# B&R Automation Studio project Nitto
Automation Studio 4.0.14.208

## Configuration Config1

CPU , AutomationRuntime G4.06, Build 4.1.2, Safety 1.5

### Task classes (Cpu.sw)
```
Cyclic#1:
  ncsdcctrl <- MainMachineCtrl.ncsdcctrl.prg
  WebControl <- (binary)
Cyclic#2:
  dummy <- MainMachineCtrl.dummy.prg
  MAIN <- MainMachineCtrl.MAIN.prg
Cyclic#4:
  VisuTasks <- Visualization.VisuCycl.VisuTasks.prg
  VisuPages <- Visualization.VisuCycl.VisuPages.prg
  VisuRange <- Visualization.VisuCycl.VisuRange.prg
  GeneralAla <- Alarme.GeneralAlarms.prg
  al_hdl <- pkgRecipe.al_hdl.prg
Cyclic#8:
  picctrl <- pkgRecipe.picctrl.prg
  tool_hdl <- pkgRecipe.tool_hdl.prg
  csv_hdl <- pkgRecipe.csv_hdl.prg
  save2USB <- pkgRecipe.save2USB.prg
DataObjects: Acp10sys
NcDataObjects: acp10etxde <- acp10etxde.dob, gunwfeedi <- AxisObj.gunwfeedi.dob, gunwfeeda <- AxisObj.gunwfeeda.dob, gmasteri <- AxisObj.gmasteri.dob, gpbs1i <- AxisObj.gpbs1i.dob, gpbs2i <- AxisObj.gpbs2i.dob, gcut1i <- AxisObj.gcut1i.dob, gcut2i <- AxisObj.gcut2i.dob, gunwopi <- AxisObj.gunwopi.dob, gunwdrvi <- AxisObj.gunwdrvi.dob, ggrid1i <- AxisObj.ggrid1i.dob, ggrid2i <- AxisObj.ggrid2i.dob, gbufferi <- AxisObj.gbufferi.dob, glongcuti <- AxisObj.glongcuti.dob, gcatchbi <- AxisObj.gcatchbi.dob, ggridfeedi <- AxisObj.ggridfeedi.dob, gconvbi <- AxisObj.gconvbi.dob, gbuffera <- AxisObj.gbuffera.dob, ggrida <- AxisObj.ggrida.dob, gunwa <- AxisObj.gunwa.dob, gpbs1a <- AxisObj.gpbs1a.dob, gpbs2a <- AxisObj.gpbs2a.dob, gcatchba <- AxisObj.gcatchba.dob, gsafetya <- AxisObj.gsafetya.dob, gconvbelta <- AxisObj.gconvbelta.dob, acp10etxd1 <- acp10etxde.dob, gPackBelta <- AxisObj.gPackBelta.dob, gPackBelti <- AxisObj.gPackBelti.dob, gCut1, gCut2, ggridfeede
VcDataObjects: Visu <- Visualization.VisuCycl.Visu.dob, Visu1 <- Visualization.VisuCycl.Visu1.dob, Visu2 <- Visualization.VisuCycl.Visu2.dob
Binaries: vcpkat, vcnet, vcpdvnc, vccpopup, vcclbox, vcctext, vccovl, vccalarm, Visu03, vccnum, vcchspot, arialbd, vccline, vccbtn, vccstr, vccddbox, vccbmp, vccshape, vccdt, vcfile, arial, vctcal, vcshared, vcrt, vcmgr, vcbclass, Visu02, vcgclass, vcdsint, vcptelo, Visu01, vcpdsw, vcpfapc, vcresman, vcpdi855, vcpdi815, vcfntttf, vcalarm, vcdsloc, vcpfmtcx, visvc, Visu103, vcpdihd, Visu102, vcpfpp50, Visu101, vcvisapi, Visu202, vcchtml, Visu201, vccurl, vcxml, Visu203, acp10cfg, acp10map, asfw, iomap, arconfig, sysconf, ashwd
Libraries: Acp10man, Acp10par, NcGlobal, UtilTyp, AsARCfg, AsBrMath, AsBrStr, AsMem, asstring, AsUSB, brsystem, FileIO, LoopConR, powerlnk, standard, sys_lib, Visapi, CSV_File, HlpStr, SwitchConf, TorqueCtrl, UserVC, Acp10_MC, Acp10sdc, SafeMC, MC_RegMa, AsMath, Acp10sim, AsWndCon, UserSpilke, SprMachine, SprManual, SprSetup, SprRegMa, SprGeneral, Runtime, AsTime, Bibliothek, dataobj, asieccon
```

### Task classes (Cpu2.sw)
```

```

### Cpu.per - 5PP5CP_US15_02/Cpu.per
```iecst
(********************************************************************
 * COPYRIGHT -- Microsoft
 ********************************************************************
 * Datei: Cpu.per
 * Autor: okrebs
 * Erstellt: 22. Mai 2014
 ********************************************************************
 * Deklaration der permanenten Variablen
 ********************************************************************)
VAR_CONFIG
	gMachRecipe AT %M0; (* *)
	gApplRecipe AT %M432; (* *)
	gPermValid AT %MD1976; (* *)
END_VAR
```

### IoMap.iom - 5PP5CP_US15_02/IoMap.iom
```iecst
(********************************************************************
 * COPYRIGHT -- Microsoft
 ********************************************************************
 * Datei: IoMap.iom
 * Autor: okrebs
 * Erstellt: 22. Mai 2014
 ********************************************************************
 * IO-Rangierungsdatei
 ********************************************************************)
VAR_CONFIG
	MAIN:machine.safety.ResetStartupInhibit AT %QX."X20SL8010_9A1".BOOL102;
	MAIN:machine.safety.ResetSafeMC AT %QX."X20SL8010_9A1".BOOL101;
	MAIN:machine.safety.ResetStartupInhibit AT %QX."X20SL8010_9A1".BOOL103;
	MAIN:machine.IOs.controlOn AT %QX."X20SL8010_9A1".BOOL104;
	MAIN:machine.safety.Control_OFF AT %QX."X20SL8010_9A1".BOOL105;
	MAIN:machine.safety.RequestSTO AT %IX."X20SL8010_9A1".BOOL001;
	MAIN:machine.safety.RequestSLS AT %IX."X20SL8010_9A1".BOOL002;
	MAIN:machine.safety.Request_ONdelay AT %IX."X20SL8010_9A1".BOOL003;
	MAIN:machine.panel.LDTControlON.LDT.button AT %IX."X20DI9371_10A6".DigitalInput01 INVERSE;
	MAIN:machine.panel.LDTControlOFF.LDT.button AT %IX."X20DI9371_10A6".DigitalInput02 INVERSE;
	MAIN:machine.panel.LDTAutomatic.LDT.button AT %IX."X20DI9371_10A6".DigitalInput03;
	MAIN:machine.panel.LDTStop.LDT.button AT %IX."X20DI9371_10A6".DigitalInput04;
	MAIN:machine.panel.LDTRESET.LDT.button AT %IX."X20DI9371_10A6".DigitalInput05;
	MAIN:machine.panel.LDTJOG.LDT.button AT %IX."X20DI9371_10A6".DigitalInput06;
	MAIN.machine.panel.LDTControlON.LDT.led AT %QX."X20DO9322_10A10".DigitalOutput01;
	MAIN.machine.panel.LDTControlOFF.LDT.led AT %QX."X20DO9322_10A10".DigitalOutput02;
	MAIN:machine.panel.LDTAutomatic.LDT.led AT %QX."X20DO9322_10A10".DigitalOutput03;
	MAIN.machine.panel.LDTStop.LDT.led AT %QX."X20DO9322_10A10".DigitalOutput04;
	MAIN:machine.panel.LDTRESET.LDT.led AT %QX."X20DO9322_10A10".DigitalOutput05;
	MAIN:machine.panel.LDTJOG.LDT.led AT %QX."X20DO9322_10A10".DigitalOutput06;
	MAIN:machine.IOs.ampel.Gruen.led AT %QX."X20DO9322_10A10".DigitalOutput09; (*MAIN.machine.IOs.ampel.Gruen.Value.ActOut*)
	MAIN:machine.IOs.ampel.Gelb.led AT %QX."X20DO9322_10A10".DigitalOutput10; (*MAIN.machine.IOs.ampel.Gelb.Value.ActOut*)
	MAIN:machine.IOs.ampel.Rot.led AT %QX."X20DO9322_10A10".DigitalOutput11; (*MAIN.machine.IOs.ampel.Rot.Value.ActOut*)
	MAIN.machine.safety.valid AT %IX."X20SO4110_10A3".PhysicalStateChannel1;
	MAIN:machine.UnwinderUnit.unwinderDrv.lift.go_up AT %QX."X20DO4332_102A8".DigitalOutput01; (*MAIN.machine.UnwinderUnit.unwinderOp.lift.go_up*)
	MAIN:machine.UnwinderUnit.unwinderOp.lift.go_up AT %QX."X20DO4332_102A8".DigitalOutput02;
	MAIN.machine.UnwinderUnit.unwinderDrv.lift.commonValve AT %QX."X20DO4332_102A8".DigitalOutput03; (*MAIN.machine.UnwinderUnit.unwinderDrv.lift.commonValve*)
	MAIN.machine.UnwinderUnit.unwinderOp.lift.commonValve AT %QX."X20DO4332_102A8".DigitalOutput04; (*MAIN.machine.UnwinderUnit.unwinderDrv.lift.commonValve*)
	MAIN.machine.UnwinderUnit.unwinderOp.lift.buttonUp AT %IX."X20DI9371_102A2".DigitalInput07; (*MAIN.machine.UnwinderUnit.unwinderOp.lift.buttonUp*)
	MAIN.machine.UnwinderUnit.unwinderOp.lift.buttonDown AT %IX."X20DI9371_102A2".DigitalInput08; (*MAIN.machine.UnwinderUnit.unwinderOp.lift.buttonDown*)
	MAIN.machine.UnwinderUnit.unwinderOp.lift.limitswitch AT %IX."X20DI9371_102A2".DigitalInput09; (*MAIN.machine.UnwinderUnit.unwinderOp.lift.limitswitch*)
	MAIN.machine.UnwinderUnit.unwinderDrv.lift.buttonUp AT %IX."X20DI9371_102A2".DigitalInput10; (*MAIN.machine.UnwinderUnit.unwinderDrv.lift.buttonUp*)
	MAIN.machine.UnwinderUnit.unwinderDrv.lift.buttonDown AT %IX."X20DI9371_102A2".DigitalInput11; (*MAIN.machine.UnwinderUnit.unwinderDrv.lift.buttonDown*)
	MAIN.machine.UnwinderUnit.unwinderDrv.lift.limitswitch AT %IX."X20DI9371_102A2".DigitalInput12; (*MAIN.machine.UnwinderUnit.unwinderDrv.lift.limitswitch*)
	MAIN:machine.IOs.hydraulicPump AT %QX."X20DO9322_10A8".DigitalOutput07;
	MAIN:machine.turngridwinder.TurnGrWinKeysbox.feederturnkey.LDT.button AT %IX."X20DI9371_202A3".DigitalInput05;
	MAIN.machine.turngridwinder.TurnGrWinKeysbox.GridWinrightkey.buttonDown.LDT.button AT %IX."X20DI9371_202A3".DigitalInput03;
	MAIN.machine.turngridwinder.TurnGrWinKeysbox.GridWinleftkey.buttonDown.LDT.button AT %IX."X20DI9371_202A3".DigitalInput04;
	MAIN.machine.turngridwinder.TurnGrWinKeysbox.GridWinrightkey.buttonDown.LDT.led AT %QX."X20DO9322_202A6".DigitalOutput09;
	MAIN.machine.turngridwinder.TurnGrWinKeysbox.GridWinleftkey.buttonDown.LDT.led AT %QX."X20DO9322_202A6".DigitalOutput10;
	MAIN:machine.ctrl.valveterminal AT %QB."X20DS4387_101A2".DataOut01_01;
	MAIN:machine.UnwinderUnit.unwinderOp.clamp.buttonDown.LDT.button AT %IX."X20DI9371_102A3".DigitalInput06;
	MAIN:machine.UnwinderUnit.unwinderOp.clamp.buttonDown.LDT.led AT %QX."X20DO9322_102A5".DigitalOutput10;
	MAIN:machine.UnwinderUnit.clamp.buttonDown.LDT.led AT %QX."X20DO9322_102A5".DigitalOutput11;
	MAIN:machine.UnwinderUnit.unwinderDrv.clamp.buttonDown.LDT.led AT %QX."X20DO9322_102A5".DigitalOutput12;
	MAIN:machine.UnwinderUnit.unwinderDrv.clamp.buttonDown.LDT.button AT %IX."X20DI9371_102A3".DigitalInput08;
	MAIN:machine.UnwinderUnit.clamp.buttonDown.LDT.button AT %IX."X20DI9371_102A3".DigitalInput07;
	MAIN:machine.UnwinderUnit.feederCtrl.LimitSwitchRight AT %IX."X20DI9371_102A3".DigitalInput04;
	MAIN:machine.UnwinderUnit.feederCtrl.LimitSwitchLeft AT %IX."X20DI9371_102A3".DigitalInput05; (*MAIN:machine.UnwinderUnit.feederCtrl.LimitSwitchLeft*)
	MAIN:machine.UnwinderUnit.feederCtrl.buttonRequestOpSide.LDT.button AT %IX."X20DI9371_102A3".DigitalInput01;
	MAIN:machine.UnwinderUnit.feederCtrl.buttonLeftOpSide.LDT.button AT %IX."X20DI9371_102A3".DigitalInput02;
	MAIN:machine.UnwinderUnit.feederCtrl.buttonRightOpSide.LDT.button AT %IX."X20DI9371_102A3".DigitalInput03;
	MAIN:machine.UnwinderUnit.feederCtrl.buttonRequestDrvSide.LDT.button AT %IX."X20DI9371_102A4".DigitalInput01;
	MAIN:machine.UnwinderUnit.feederCtrl.buttonRightDrvSide.LDT.button AT %IX."X20DI9371_102A4".DigitalInput02;
	MAIN:machine.UnwinderUnit.feederCtrl.buttonLeftDrvSide.LDT.button AT %IX."X20DI9371_102A4".DigitalInput03;
	Cyclic#1.gUnwFeeder_DrvIf.iDrvOK AT %IX."8I64xxxxxxx.00x-1".ETAD_Input_Bool_02;
	Cyclic#1.gUnwFeeder_DiDoIf.iDriveReady AT %IX."8I64xxxxxxx.00x-1".ETAD_Input_Bool_02;
	Cyclic#1.gUnwFeeder_ModuleOk AT %IX."8I64xxxxxxx.00x-1".ModuleOk;
	Cyclic#1.gUnwFeeder_DrvIf.iLifeCnt AT %IB."8I64xxxxxxx.00x-1".SDC_LifeCnt;
	Cyclic#1.gUnwFeeder_DiDoIf.iLifeCntDriveEnable AT %IB."8I64xxxxxxx.00x-1".SDC_LifeCnt;
	Cyclic#1.gUnwFeeder_DiDoIf.iLifeCntDriveReady AT %IB."8I64xxxxxxx.00x-1".SDC_LifeCnt;
	Cyclic#1.gUnwFeeder_DiDoIf.oDriveEnable AT %QX."8I64xxxxxxx.00x-1".CMDD_Output_Bool_00;
	Cyclic#1.gUnwFeeder_ModuleOk AT %QX."8I64xxxxxxx.00x-1".CMDD_Output_Bool_01;
	Cyclic#1.gUnwFeeder_ModuleOk AT %QX."8I64xxxxxxx.00x-1".CMDD_Output_Bool_02;
	Cyclic#1.gUnwFeeder_DiDoIf.oDriveEnable AT %QX."8I64xxxxxxx.00x-1".CMDD_Output_Bool_03;
	Cyclic#1.gUnwFeeder_DrvIf.oSetPos AT %QW."8I64xxxxxxx.00x-1".LFRD_Output;
	Cyclic#1.gUnwFeeder_DrvIf.oSetTime AT %QW."8I64xxxxxxx.00x-1".SDC_SetTime;
	Cyclic#1.gUnwFeeder_DrvIf.oBrake AT %QX."8I64xxxxxxx.00x-1".DigitalOutput01;
	MAIN:machine.turngridwinder.TurnGrWinKeysbox.feederturnkey.LDT.led AT %QX."X20DO9322_202A6".DigitalOutput11;
	::MAIN:machine.UnwinderUnit.splicetable.clampAfter.buttonDown.LDT.button AT %IX."X20DI9371_102A3".DigitalInput09; (*MAIN:machine.UnwinderUnit.splicetable.clampBefore.buttonDown.LDT.button*)
	::MAIN:machine.UnwinderUnit.splicetable.clampBefore.buttonDown.LDT.button AT %IX."X20DI9371_102A4".DigitalInput08; (*MAIN:machine.UnwinderUnit.splicetable.clampAfter.buttonDown.LDT.button*)
	MAIN:machine.UnwinderUnit.unwinderOp.lift.LED_is_up AT %QX."X20DO9322_102A5".DigitalOutput05;
	MAIN:machine.UnwinderUnit.unwinderOp.lift.go_up AT %QX."X20DO9322_102A5".DigitalOutput06;
	MAIN:machine.UnwinderUnit.unwinderDrv.lift.LED_is_up AT %QX."X20DO9322_102A5".DigitalOutput07;
	MAIN:machine.UnwinderUnit.unwinderDrv.lift.go_up AT %QX."X20DO9322_102A5".DigitalOutput08;
	::MAIN:machine.UnwinderUnit.splicetable.clampAfter.buttonDown.LDT.led AT %QX."X20DO9322_102A6".DigitalOutput01;
	MAIN:machine.pullbreak.clamp.buttonDown.LDT.button AT %IX."X20DI9371_102A3".DigitalInput11;
	::MAIN:machine.UnwinderUnit.splicetable.clampBefore.buttonDown.LDT.led AT %QX."X20DO9322_102A6".DigitalOutput06;
	MAIN:machine.safety.manuelmode AT %QX."X20SL8010_9A1".BOOL106;
	MAIN:machine.webguidingbuffer.active AT %QX."X20DO9322_10A9".DigitalOutput01;
	MAIN:machine.webguidingbuffer.handSelect AT %QX."X20DO9322_10A9".DigitalOutput02;
	MAIN:machine.webguidingbuffer.neutral AT %QX."X20DO9322_10A9".DigitalOutput03;
	MAIN:machine.webguidingbuffer.automatic AT %QX."X20DO9322_10A9".DigitalOutput04;
	MAIN:machine.webguidingbuffer.arrowLeft AT %QX."X20DO9322_10A9".DigitalOutput05;
	MAIN:machine.webguidingbuffer.arrowRight AT %QX."X20DO9322_10A9".DigitalOutput06;
	MAIN:machine.webguiding.active AT %QX."X20DO9322_10A9".DigitalOutput07;
	MAIN:machine.webguiding.manual AT %QX."X20DO9322_10A9".DigitalOutput08;
	MAIN:machine.webguiding.neutral AT %QX."X20DO9322_10A9".DigitalOutput09;
	MAIN:machine.webguiding.automatic AT %QX."X20DO9322_10A9".DigitalOutput10;
	MAIN:machine.webguiding.arrowLeft AT %QX."X20DO9322_10A9".DigitalOutput11;
	MAIN:machine.webguiding.arrowRight AT %QX."X20DO9322_10A9".DigitalOutput12;
	MAIN:machine.summerystartstop.boxunwinder.start.LDT.button AT %IX."X20DI9371_102A2".DigitalInput01;
	MAIN:machine.summerystartstop.boxunwinder.stop.LDT.button AT %IX."X20DI9371_102A2".DigitalInput02;
	MAIN:machine.summerystartstop.boxunwinder.jog.LDT.button AT %IX."X20DI9371_102A2".DigitalInput03;
	MAIN:machine.summerystartstop.boxwebbuffer.start.LDT.button AT %IX."X20DI9371_102A2".DigitalInput04;
	MAIN:machine.summerystartstop.boxwebbuffer.stop.LDT.button AT %IX."X20DI9371_102A2".DigitalInput05;
	MAIN:machine.summerystartstop.boxwebbuffer.jog.LDT.button AT %IX."X20DI9371_102A2".DigitalInput06;
	MAIN:machine.summerystartstop.boxcutting1.start.LDT.button AT %IX."X20DI9371_202A2".DigitalInput01;
	MAIN:machine.summerystartstop.boxcutting1.stop.LDT.button AT %IX."X20DI9371_202A2".DigitalInput02;
	MAIN:machine.summerystartstop.boxcutting1.jog.LDT.button AT %IX."X20DI9371_202A2".DigitalInput03;
	MAIN:machine.cuttingunit1.powerbridge.bridgedownbutton.buttonDown.LDT.button AT %IX."X20DI9371_202A2".DigitalInput07;
	MAIN:machine.cuttingunit2.powerbridge.bridgedownbutton.buttonDown.LDT.button AT %IX."X20DI9371_202A2".DigitalInput11;
	MAIN:machine.longcutter.cutterUp.buttomToggle.LDT.button AT %IX."X20DI9371_202A3".DigitalInput09; (*MAIN:machine.longcutter.cutterUp.buttomToggle.LDT.button*)
	MAIN:machine.longcutter.discmovesupp.buttonDown.LDT.button AT %IX."X20DI9371_202A3".DigitalInput10; (*MAIN:machine.longcutter.discmovesupp.buttonDown.LDT.button*)
	MAIN:machine.pullbreakSt.hubctrl.buttomToggle2.LDT.button AT %IX."X20DI9371_202A4".DigitalInput04; (*MAIN:machine.pullbreakSt.hubctrl.buttomToggle2.LDT.button*)
	MAIN:machine.summerystartstop.boxconveyor.start.LDT.button AT %IX."X20DI9371_202A5".DigitalInput03;
	MAIN:machine.summerystartstop.boxconveyor.stop.LDT.button AT %IX."X20DI9371_202A5".DigitalInput04;
	MAIN:machine.summerystartstop.boxconveyor.jog.LDT.button AT %IX."X20DI9371_202A5".DigitalInput05;
	MAIN:machine.summerystartstop.boxlongcutter.jog.LDT.button AT %IX."X20DI9371_202A3".DigitalInput11; (*MAIN:machine.longcutter.movebutton.LDT.button*)
	MAIN:machine.cuttingunit2.powerbridge.movebutton.LDT.button AT %IX."X20DI9371_202A2".DigitalInput12;
	MAIN:machine.cuttingunit1.powerbridge.movebutton.LDT.button AT %IX."X20DI9371_202A2".DigitalInput08;
	MAIN:machine.cuttingunit1.axis.refSwitchConfig.HomeSwitch AT %IX."X20DI9371_202A2".DigitalInput09 INVERSE;
	MAIN:machine.cuttingunit2.axis.refSwitchConfig.HomeSwitch AT %IX."X20DI9371_202A3".DigitalInput01 INVERSE;
	MAIN:machine.IOs.ValveAirON AT %QX."X20DO9322_202A11".DigitalOutput01;
	MAIN:machine.pullbreak.clamp.buttonDown.LDT.led AT %QX."X20DO9322_102A6".DigitalOutput02;
	MAIN:machine.ctrl.valveterminal2 AT %QB."X20DS4387_101A2".DataOut02_01;
	MAIN:machine.ctrl.valveterminal22 AT %QB."X20DS4387_101A2".DataOut02_02;
	MAIN:machine.cuttingunit1.powerbridge.bridgedownbutton.buttonDown.LDT.led AT %QX."X20DO9322_202A6".DigitalOutput05;
	MAIN:machine.cuttingunit2.powerbridge.bridgedownbutton.buttonDown.LDT.led AT %QX."X20DO9322_202A6".DigitalOutput07;
	MAIN:machine.longcutter.cutterUp.buttomToggle.LDT.ledinv AT %QX."X20DO9322_202A6".DigitalOutput12;
	MAIN:machine.pullbreakSt.hubctrl.buttomToggle.LDT.button AT %IX."X20DI9371_202A4".DigitalInput05; (*MAIN:machine.pullbreakSt.hubctrl.buttomToggle.LDT.button*)
	MAIN:machine.longcutter.discmovesupp.buttonDown.LDT.led AT %QX."X20DO9322_202A7".DigitalOutput01;
	MAIN:machine.longcutter.cutterUp.isup AT %IX."X20DI9371_202A3".DigitalInput07;
	MAIN:machine.pullbreakSt.hubctrl.isdown AT %IX."X20DI9371_202A4".DigitalInput01; (*MAIN:machine.pullbreakSt.hubctrl.isdown*)
	MAIN:machine.pullbreakSt.hubctrl.isup AT %IX."X20DI9371_202A3".DigitalInput12; (*MAIN:machine.pullbreakSt.hubctrl.isup*)
	Cyclic#1.gUnwFeeder_DiDoIf.oDriveEnable AT %QX."8I64xxxxxxx.00x-1".CMDD_Output_Bool_07;
	MAIN:machine.webbuffer.axis.refSwitchConfig.NegHWSwitch AT %IX."X20DI9371_102A4".DigitalInput07 INVERSE;
	MAIN:machine.webbuffer.axis.refSwitchConfig.PosHWSwitch AT %IX."X20DI9371_102A4".DigitalInput06 INVERSE;
	MAIN:machine.ctrl.valveterminal23 AT %QB."X20DS4387_101A2".DataOut02_03;
	MAIN:machine.switchcabinet.EMCY_Buttons.EMCY_Button1 AT %IX."X20SI4100_10A1".SafeEquivalentInput0102; (*Schaltschrank*)
	MAIN:machine.panel.EMCY_Button AT %IX."X20SI4100_10A1".SafeEquivalentInput0304; (*Panel*)
	MAIN:machine.cuttingunit1.powerbridge.pressuredrvside AT %IW."X20AI4622_202A8".AnalogInput01;
	MAIN:machine.cuttingunit1.powerbridge.pressureOperside AT %IW."X20AI4622_202A8".AnalogInput02;
	MAIN:machine.cuttingunit2.powerbridge.pressuredrvside AT %IW."X20AI4622_202A8".AnalogInput03; (*MAIN:machine.cuttingunit2.powerbridge.pressureOperside*)
	MAIN:machine.cuttingunit2.powerbridge.pressureOperside AT %IW."X20AI4622_202A8".AnalogInput04;
	MAIN:machine.UnwinderUnit.emcy_inputs.EMCY_Button1 AT %IX."X20SI9100_101A3".SafeTwoChannelInput0102;
	MAIN:machine.emcy_inputs.EMCY_Button1 AT %IX."X20SI9100_101A3".SafeTwoChannelInput0304;
	MAIN:machine.UnwinderUnit.emcy_inputs.EMCY_Button2 AT %IX."X20SI9100_101A3".SafeTwoChannelInput0506;
	MAIN:machine.emcy_inputs.EMCY_pullwireOPs AT %IX."X20SI9100_101A3".SafeTwoChannelInput0708;
	MAIN:machine.emcy_inputs.EMCY_pullwireDVRs AT %IX."X20SI9100_101A3".SafeTwoChannelInput0910;
	MAIN:machine.webbuffer.emcy_inputs.EMCY_Door1 AT %IX."X20SI9100_101A3".SafeTwoChannelInput1112;
	MAIN:machine.webbuffer.emcy_inputs.EMCY_Door2 AT %IX."X20SI9100_101A3".SafeTwoChannelInput1516;
	MAIN:machine.webbuffer.emcy_inputs.EMCY_Door6 AT %IX."X20SI9100_101A3".SafeTwoChannelInput1718;
	MAIN:machine.webbuffer.emcy_inputs.EMCY_Door3 AT %IX."X20SI9100_101A3".SafeTwoChannelInput1920;
	MAIN:machine.webbuffer.emcy_inputs.EMCY_Door4 AT %IX."X20SI9100_101A4".SafeTwoChannelInput0102;
	MAIN:machine.webbuffer.emcy_inputs.EMCY_Door5 AT %IX."X20SI9100_101A4".SafeTwoChannelInput0304;
	MAIN:machine.pullbreak.emcy_inputs.EMCY_Door1 AT %IX."X20SI9100_101A4".SafeTwoChannelInput0910;
	MAIN:machine.emcy_inputs.EMCY_Button2 AT %IX."X20SI9100_201A2".SafeTwoChannelInput0102;
	MAIN:machine.emcy_inputs.EMCY_Button4 AT %IX."X20SI9100_201A2".SafeTwoChannelInput0304;
	MAIN:machine.emcy_inputs.EMCY_Button3 AT %IX."X20SI9100_201A2".SafeTwoChannelInput0506;
	MAIN:machine.cuttingunit1.emcy_inputs.EMCY_Door1 AT %IX."X20SI9100_201A2".SafeTwoChannelInput0708;
	MAIN:machine.cuttingunit1.emcy_inputs.EMCY_Door2 AT %IX."X20SI9100_201A2".SafeTwoChannelInput0910;
	MAIN:machine.cuttingunit2.emcy_inputs.EMCY_Door1 AT %IX."X20SI9100_201A2".SafeTwoChannelInput1112;
	MAIN:machine.cuttingunit2.emcy_inputs.EMCY_Door2 AT %IX."X20SI9100_201A2".SafeTwoChannelInput1314;
	MAIN:machine.longcutter.emcy_inputs.EMCY_Door1 AT %IX."X20SI9100_201A2".SafeTwoChannelInput1516;
	MAIN:machine.conveyor.emcy_inputs.EMCY_Button2 AT %IX."X20SI9100_201A2".SafeTwoChannelInput1718;
	MAIN:machine.conveyor.emcy_inputs.EMCY_Button1 AT %IX."X20SI9100_201A2".SafeTwoChannelInput1920;
	MAIN:machine.pullbreakSt.hubctrl.limiterSwitchDrvSide AT %IX."X20DI9371_202A4".DigitalInput03; (*MAIN:machine.pullbreakSt.hubctrl.limiterSwitchDrvSide*)
	MAIN:machine.pullbreakSt.hubctrl.limiterSwitchOpSide AT %IX."X20DI9371_202A5".DigitalInput08;
	MAIN:machine.longcutter.cutterUp.enable AT %IX."X20DI9371_202A3".DigitalInput06 INVERSE;
	MAIN:machine.conveyor.counters.counter1.triggerInput AT %IX."X20DI9371_202A4".DigitalInput06;
	MAIN:machine.conveyor.counters.counter2.triggerInput AT %IX."X20DI9371_202A4".DigitalInput07;
	MAIN:machine.conveyor.counters.counter3.triggerInput AT %IX."X20DI9371_202A4".DigitalInput08;
	MAIN:machine.conveyor.counters.counter4.triggerInput AT %IX."X20DI9371_202A4".DigitalInput09;
	MAIN:machine.conveyor.counters.counter5.triggerInput AT %IX."X20DI9371_202A4".DigitalInput10;
	MAIN:machine.conveyor.counters.counter6.triggerInput AT %IX."X20DI9371_202A4".DigitalInput11;
	MAIN:machine.conveyor.counters.counter7.triggerInput AT %IX."X20DI9371_202A4".DigitalInput12;
	MAIN:machine.conveyor.counters.counter8.triggerInput AT %IX."X20DI9371_202A5".DigitalInput01;
	MAIN:machine.conveyor.counters.counter9.triggerInput AT %IX."X20DI9371_202A5".DigitalInput02;
	MAIN:machine.conveyor.counters.reset AT %IX."X20DI9371_202A5".DigitalInput06;
	MAIN:machine.switchcabinet.fusePlug1 AT %IX."X20DI9371_10A5".DigitalInput01;
	MAIN:machine.switchcabinet.fusePlug2 AT %IX."X20DI9371_10A5".DigitalInput02;
	MAIN:machine.switchcabinet.fusePlugCEE AT %IX."X20DI9371_10A5".DigitalInput03;
	MAIN:machine.switchcabinet.aircond AT %IX."X20DI9371_10A5".DigitalInput04;
	MAIN:machine.switchcabinet.fuseWebGuide1 AT %IX."X20DI9371_10A5".DigitalInput05;
	MAIN:machine.webguidingbuffer.hardwareOK AT %IX."X20DI9371_10A5".DigitalInput06;
	MAIN:machine.switchcabinet.fuseWebGuide2 AT %IX."X20DI9371_10A5".DigitalInput07;
	MAIN:machine.webguiding.hardwareOK AT %IX."X20DI9371_10A5".DigitalInput08;
	MAIN:machine.longcutter.webclamp.buttonDown.LDT.button AT %IX."X20DI9371_202A3".DigitalInput02;
	MAIN:machine.longcutter.webclamp.toDown_o AT %QX."X20DO9322_202A7".DigitalOutput08;
	MAIN:machine.webbuffer.keys.up.LDT.button AT %IX."X20DI9371_102A4".DigitalInput09;
	MAIN:machine.webbuffer.keys.down.LDT.button AT %IX."X20DI9371_102A4".DigitalInput10;
	MAIN:machine.webbuffer.keys.home.LDT.button AT %IX."X20DI9371_102A4".DigitalInput11;
	MAIN:machine.webbuffer.keys.up.LDT.led AT %QX."X20DO9322_102A6".DigitalOutput07;
	MAIN:machine.webbuffer.keys.down.LDT.led AT %QX."X20DO9322_102A6".DigitalOutput08;
	MAIN:machine.webbuffer.keys.home.LDT.led AT %QX."X20DO9322_102A6".DigitalOutput09;
	MAIN:machine.masterModul.ctrl.handWheel.counterHandWheel AT %IW."X20DC1196_202A9".Encoder01;
	MAIN:OutputGrinderON AT %QX."X20DO9322_10A8".DigitalOutput05;
	MAIN:machine.IOs.ampel.horn_o AT %QX."X20DO9322_10A10".DigitalOutput12;
	MAIN:machine.UnwinderUnit.feederCtrl.buttonRequestOpSide.LDT.led AT %QX."X20DO9322_102A5".DigitalOutput09;
	MAIN:machine.UnwinderUnit.feederCtrl.buttonRequestDrvSide.LDT.led AT %QX."X20DO9322_102A6".DigitalOutput05;
	MAIN:machine.masterModul.ctrl.inlineVelocity.dancepos AT %IW."X20AI4622_101A5".AnalogInput01;
	MAIN:machine.panel.LDTAutomatic.LDT.led AT %QX."X20DO9322_10A10".DigitalOutput07;
	MAIN:machine.IOs.antistatik AT %QX."X20DO9322_10A8".DigitalOutput01;
	MAIN:machine.IOs.inline AT %QX."X20DO9322_10A8".DigitalOutput08;
	MAIN:machine.IOs.machineReady AT %QX."X20DO9322_10A8".DigitalOutput09;
	MAIN:machine.masterModul.ctrl.inlineVelocity.ConveyerVelocity AT %IW."X20AI4622_10A12".AnalogInput01;
	::MAIN:machine.webbuffer.dancer.FlengeDMS AT %QB."X20AI1744_101A6".ConfigOutput01;
	::MAIN:machine.webbuffer.dancer.DMS_In AT %ID."X20AI1744_101A6".AnalogInput01;
	::MAIN:machine.conveyor.counters.Nitto_Table_Full AT %QX."X20DO9322_202A11".DigitalOutput02;
	::MAIN:machine.IOs.Unwinder_OP_Led AT %QX."X20DO9322_202A6".DigitalOutput03;
	::MAIN:machine.IOs.Unwinder_Drv_Led AT %QX."X20DO9322_202A6".DigitalOutput04;
	::MAIN:machine.IOs.Unwinder_Drv_Button AT %IX."X20DI9371_202A2".DigitalInput04;
	::MAIN:machine.IOs.Unwinder_OP_Button AT %IX."X20DI9371_202A2".DigitalInput05;
	::MAIN:machine.ctrl.tasktimerPos AT %QX."X20DO9322_10A8".DigitalOutput11;
	::MAIN:machine.ctrl.tasktimerNeg AT %QX."X20DO9322_10A8".DigitalOutput12;
	Cyclic#1.gPackBelt_DrvIf.iLifeCnt AT %IB."8I64xxxxxxx.00x-1a".SDC_LifeCnt;
	Cyclic#1.gPackBelt_DrvIf.iDrvOK AT %IX."8I64xxxxxxx.00x-1a".ETAD_Input_Bool_02;
	Cyclic#1.gPackBelt_DrvIf.oSetTime AT %QW."8I64xxxxxxx.00x-1a".SDC_SetTime;
	Cyclic#1.gPackBelt_DrvIf.oSetPos AT %QW."8I64xxxxxxx.00x-1a".LFRD_Output;
	Cyclic#1.gPackBelt_DiDoIf.iLifeCntDriveReady AT %IB."8I64xxxxxxx.00x-1a".SDC_LifeCnt;
	Cyclic#1.gPackBelt_DiDoIf.iLifeCntDriveEnable AT %IB."8I64xxxxxxx.00x-1a".SDC_LifeCnt;
	Cyclic#1.gPackBelt_DiDoIf.oDriveEnable AT %QX."8I64xxxxxxx.00x-1a".CMDD_Output_Bool_00;
	Cyclic#1.gPackBelt_ModuleOk AT %QX."8I64xxxxxxx.00x-1a".CMDD_Output_Bool_01;
	Cyclic#1.gPackBelt_ModuleOk AT %QX."8I64xxxxxxx.00x-1a".CMDD_Output_Bool_02;
	Cyclic#1.gPackBelt_ModuleOk AT %IX."8I64xxxxxxx.00x-1a".ModuleOk;
	Cyclic#1.gPackBelt_DiDoIf.oDriveEnable AT %QX."8I64xxxxxxx.00x-1a".CMDD_Output_Bool_03;
	Cyclic#1.gPackBelt_DiDoIf.iDriveReady AT %IX."8I64xxxxxxx.00x-1a".ETAD_Input_Bool_02;
	Cyclic#1.gPackBelt_DiDoIf.oDriveEnable AT %QX."8I64xxxxxxx.00x-1a".CMDD_Output_Bool_07;
	Cyclic#1.gPackBelt_DrvIf.oBrake AT %QX."8I64xxxxxxx.00x-1a".DigitalOutput01;
	MAIN:machine.turngridwinder.ctrl.refSwitchConfig.HomeSwitch AT %IX."X20DI9371_202A3".DigitalInput08;
	::MAIN:machine.conveyor.emcy_inputs.EMCY_Button3 AT %IX."X20SI4100_201A3".SafeEquivalentInput0102;
	MAIN:machine.packbelt.ctrl.switchAutomatic AT %IX."X20DI9371_202A5".DigitalInput10;
	MAIN:machine.packbelt.ctrl.switchManual AT %IX."X20DI9371_202A5".DigitalInput11;
	MAIN:machine.packbelt.ctrl.buttonStart AT %IX."X20DI9371_202A5".DigitalInput12;
	MAIN:machine.packbelt.ctrl.sensorBoxesPresent AT %IX."X20DI9371_202A5".DigitalInput09;
	MAIN:machine.packbelt.ctrl.sensorStop AT %IX."X20DI9371_202A2".DigitalInput06;
	MAIN:machine.packbelt.ctrl.sensorLowerSpeed AT %IX."X20DI9371_202A2".DigitalInput10;
	::MAIN:machine.conveyor.counters.GreenLampOut AT %QX."X20DO9322_202A11".DigitalOutput03;
	::MAIN:machine.conveyor.counters.RedLampOut AT %QX."X20DO9322_202A11".DigitalOutput04;
	::MAIN:machine.IOs.aIn.Dancer_position.Value.RawInt AT %IW."X20AI4622_101A5".AnalogInput02;
	::gMachine.IO.DIn.Liner_detekce.Value.State AT %IX."X20DI9371_102A3".DigitalInput10;
END_VAR
```

### Acp10cfg.ncc - 5PP5CP_US15_02/Motion/Acp10cfg.ncc
```
NcConfiguration (Version=2.37.0, NcSwId=Acp10)
  ACP10CF1_typ:
    cnt_nettrc_rec_drive = 1500
    bufsize_trace_upload = 1200
    tc_nc_man_task = Cyclic #1
    glob_pv_as_ncobject = Yes
    ncsys_dl_broadcast = Yes
    ncsys_dl_acp_reset = Yes
    network_init:
      ncsw_init_execute = Yes
      automatic_execute = No
      node_nr_warning = Yes
      net_err_before_ncact = Yes
    nettrc:
      enter_parsecrec = Yes
      enter_ncaction = Yes
      save_ring_startidx = Yes
    plk_if[0]:
      if_name = SL1.IF1
      tc_CycDat_PLCopen = Task class for NC Manager task
      mc_broadcast_extdat = No
    sdc_if[0]:
      if_name = SDC_IF1
      mc_broadcast_size = 800
      mc_broadcast_extdat = No
```

### Acp10map.ncm - 5PP5CP_US15_02/Motion/Acp10map.ncm
```
NcMapping (NcSwId=Acp10)
  NcObject gUnwOp (ModuleId=8BVI0110HWD0.000-1_Hauptabrollung1und2, Type=ncAXIS, Channel=1, AcoposSimulation=Off, InitParameter=gunwopi, AcoposParameter=gunwa, AdditionalData=PLCopen_ModPos="1000000,1", Disabled=FALSE, ModuleDisabled=FALSE)  // Operator side
  NcObject gUnwDrv (ModuleId=8BVI0110HWD0.000-1_Hauptabrollung1und2, Type=ncAXIS, Channel=2, AcoposSimulation=Off, InitParameter=gunwdrvi, AcoposParameter=gunwa, AdditionalData=PLCopen_ModPos="1000000,1", Disabled=FALSE, ModuleDisabled=FALSE)  // Drive side
  NcObject gCut2 (ModuleId=8BVI0330HWSS.000-1_Stanzstation2, Type=ncAXIS, Channel=1, AcoposSimulation=Off, InitParameter=gcut2i, AcoposParameter=gsafetya, AdditionalData=PLCopen_ModPos="1000000,1", Disabled=FALSE, ModuleDisabled=FALSE)
  NcObject gGridFeeder (ModuleId=8BVI0110HWSS.000-1_GitterDrehfunktion, Type=ncAXIS, Channel=1, AcoposSimulation=Off, InitParameter=ggridfeedi, AcoposParameter=gsafetya, AdditionalData=PLCopen_ModPos="360000,1", Disabled=FALSE, ModuleDisabled=FALSE)
  NcObject gCut1 (ModuleId=8BVI0330HWSS.000-1_Stanzstation1, Type=ncAXIS, Channel=1, AcoposSimulation=Off, InitParameter=gcut1i, AcoposParameter=gsafetya, AdditionalData=PLCopen_ModPos="1000000,1", Disabled=FALSE, ModuleDisabled=FALSE)
  NcObject gLongCut (ModuleId=8BVI0014HWSS.000-1_Laengsschneider, Type=ncAXIS, Channel=1, AcoposSimulation=Off, InitParameter=glongcuti, AcoposParameter=gsafetya, AdditionalData=PLCopen_ModPos="1000000,1", Disabled=FALSE, ModuleDisabled=FALSE)
  NcObject gPBS1 (ModuleId=8BVI0110HWD0.000-1_Bahnpuffer_Zugstation1, Type=ncAXIS, Channel=2, AcoposSimulation=Off, InitParameter=gpbs1i, AcoposParameter=gpbs2a, AdditionalData=PLCopen_ModPos="1000000,1", Disabled=FALSE, ModuleDisabled=FALSE)
  NcObject gPBS2 (ModuleId=8BVI0055HWD0.000-1_Zugband_Auslageband, Type=ncAXIS, Channel=1, AcoposSimulation=Off, InitParameter=gpbs2i, AcoposParameter=gpbs2a, AdditionalData=PLCopen_ModPos="1000000,1", Disabled=FALSE, ModuleDisabled=FALSE)
  NcObject gGridRight (ModuleId=8BVI0110HWD0.000-1_Gitteraufrollung1und2, Type=ncAXIS, Channel=2, AcoposSimulation=Off, InitParameter=ggrid2i, AcoposParameter=ggrida, AdditionalData=PLCopen_ModPos="1000000,1", Disabled=FALSE, ModuleDisabled=FALSE)
  NcObject gGridLeft (ModuleId=8BVI0110HWD0.000-1_Gitteraufrollung1und2, Type=ncAXIS, Channel=1, AcoposSimulation=Off, InitParameter=ggrid1i, AcoposParameter=ggrida, AdditionalData=PLCopen_ModPos="1000000,1", Disabled=FALSE, ModuleDisabled=FALSE)
  NcObject gConvBelt (ModuleId=8BVI0055HWD0.000-1_Zugband_Auslageband, Type=ncAXIS, Channel=2, AcoposSimulation=Off, InitParameter=gconvbi, AcoposParameter=gconvbelta, AdditionalData=PLCopen_ModPos="1000000,1", Disabled=FALSE, ModuleDisabled=FALSE)
  NcObject gCatchBelt (ModuleId=8BVI0014HWD0.000-1_Fangband, Type=ncAXIS, Channel=1, AcoposSimulation=Off, InitParameter=gcatchbi, AcoposParameter=gcatchba, AdditionalData=PLCopen_ModPos="1000000,1", Disabled=FALSE, ModuleDisabled=FALSE)
  NcObject gBuffer (ModuleId=8BVI0110HWD0.000-1_Bahnpuffer_Zugstation1, Type=ncAXIS, Channel=1, AcoposSimulation=Off, InitParameter=gbufferi, AcoposParameter=gbuffera, Disabled=FALSE, ModuleDisabled=FALSE)
  NcObject 8BVI0014HWSS.000-1_ncV_AXIS1 (ModuleId=8BVI0014HWSS.000-1_Laengsschneider, Type=ncV_AXIS, Channel=1, Disabled=TRUE, ModuleDisabled=FALSE)
  NcObject 8BVI0014HWD0.000-1_ncV_AXIS1 (ModuleId=8BVI0014HWD0.000-1_Fangband, Type=ncV_AXIS, Channel=1, Disabled=TRUE, ModuleDisabled=FALSE)
  NcObject 8BVI0110HWSS.000-1_ncV_AXIS1 (ModuleId=8BVI0110HWSS.000-1_GitterDrehfunktion, Type=ncV_AXIS, Channel=1, Disabled=TRUE, ModuleDisabled=FALSE)
  NcObject 8BVI0014HWSS.000-1_ncV_AXIS2 (ModuleId=8BVI0014HWSS.000-1_Laengsschneider, Type=ncV_AXIS, Channel=2, Disabled=TRUE, ModuleDisabled=FALSE)
  NcObject 8BVI0110HWSS.000-1_ncV_AXIS2 (ModuleId=8BVI0110HWSS.000-1_GitterDrehfunktion, Type=ncV_AXIS, Channel=2, Disabled=TRUE, ModuleDisabled=FALSE)
  NcObject 8BVI0014HWSS.000-1_ncAXIS2 (ModuleId=8BVI0014HWSS.000-1_Laengsschneider, Type=ncAXIS, Channel=2, AcoposSimulation=Off, Disabled=TRUE, ModuleDisabled=FALSE)
  NcObject 8BVI0014HWD0.000-1_ncAXIS2 (ModuleId=8BVI0014HWD0.000-1_Fangband, Type=ncAXIS, Channel=2, AcoposSimulation=Off, Disabled=TRUE, ModuleDisabled=FALSE)
  NcObject 8BVI0055HWD0.000-1_ncV_AXIS1 (ModuleId=8BVI0055HWD0.000-1_Zugband_Auslageband, Type=ncV_AXIS, Channel=1, Disabled=TRUE, ModuleDisabled=FALSE)
  NcObject 8BVI0110HWSS.000-1_ncAXIS2 (ModuleId=8BVI0110HWSS.000-1_GitterDrehfunktion, Type=ncAXIS, Channel=2, AcoposSimulation=Off, Disabled=TRUE, ModuleDisabled=FALSE)
  NcObject 8BVI0110HWD0.000-1b_ncV_AXIS2 (ModuleId=8BVI0110HWD0.000-1_Gitteraufrollung1und2, Type=ncV_AXIS, Channel=2, Disabled=TRUE, ModuleDisabled=FALSE)
  NcObject 8BVI0110HWD0.000-1b_ncV_AXIS1 (ModuleId=8BVI0110HWD0.000-1_Gitteraufrollung1und2, Type=ncV_AXIS, Channel=1, Disabled=TRUE, ModuleDisabled=FALSE)
  NcObject 8BVI0110HWD0.000-1a_ncV_AXIS2 (ModuleId=8BVI0110HWD0.000-1_Bahnpuffer_Zugstation1, Type=ncV_AXIS, Channel=2, Disabled=TRUE, ModuleDisabled=FALSE)
  NcObject 8BVI0110HWD0.000-1a_ncV_AXIS1 (ModuleId=8BVI0110HWD0.000-1_Bahnpuffer_Zugstation1, Type=ncV_AXIS, Channel=1, Disabled=TRUE, ModuleDisabled=FALSE)
  NcObject 8BVI0014HWD0.000-1_ncV_AXIS2 (ModuleId=8BVI0014HWD0.000-1_Fangband, Type=ncV_AXIS, Channel=2, Disabled=TRUE, ModuleDisabled=FALSE)
  NcObject 8BVI0110HWD0.000-1_ncV_AXIS2 (ModuleId=8BVI0110HWD0.000-1_Hauptabrollung1und2, Type=ncV_AXIS, Channel=2, Disabled=TRUE, ModuleDisabled=FALSE)
  NcObject 8BVI0110HWD0.000-1_ncV_AXIS1 (ModuleId=8BVI0110HWD0.000-1_Hauptabrollung1und2, Type=ncV_AXIS, Channel=1, Disabled=TRUE, ModuleDisabled=FALSE)
  NcObject 8BVI0330HWSS.000-1a_ncAXIS2 (ModuleId=8BVI0330HWSS.000-1_Stanzstation2, Type=ncAXIS, Channel=2, AcoposSimulation=Off, Disabled=TRUE, ModuleDisabled=FALSE)
  NcObject 8B0P0440HW00.000-1a_ncAXIS2 (ModuleId=8B0P0440HW00.000-1_Versorgung2, Type=ncAXIS, Channel=2, AcoposSimulation=Off, Disabled=TRUE, ModuleDisabled=FALSE)
  NcObject 8BVI0330HWSS.000-1a_ncV_AXIS2 (ModuleId=8BVI0330HWSS.000-1_Stanzstation2, Type=ncV_AXIS, Channel=2, Disabled=TRUE, ModuleDisabled=FALSE)
  NcObject 8BVI0330HWSS.000-1_ncV_AXIS1 (ModuleId=8BVI0330HWSS.000-1_Stanzstation1, Type=ncV_AXIS, Channel=1, Disabled=TRUE, ModuleDisabled=FALSE)
  NcObject 8BVI0330HWSS.000-1_ncV_AXIS2 (ModuleId=8BVI0330HWSS.000-1_Stanzstation1, Type=ncV_AXIS, Channel=2, Disabled=TRUE, ModuleDisabled=FALSE)
  NcObject 8BVI0330HWSS.000-1a_ncV_AXIS1 (ModuleId=8BVI0330HWSS.000-1_Stanzstation2, Type=ncV_AXIS, Channel=1, Disabled=TRUE, ModuleDisabled=FALSE)
  NcObject 8B0P0440HW00.000-1_ncAXIS1 (ModuleId=8B0P0440HW00.000-1_Versorgung1, Type=ncAXIS, Channel=1, AcoposSimulation=Off, Disabled=TRUE, ModuleDisabled=FALSE)
  NcObject 8B0P0440HW00.000-1a_ncV_AXIS2 (ModuleId=8B0P0440HW00.000-1_Versorgung2, Type=ncV_AXIS, Channel=2, Disabled=TRUE, ModuleDisabled=FALSE)
  NcObject 8B0P0440HW00.000-1_ncV_AXIS2 (ModuleId=8B0P0440HW00.000-1_Versorgung1, Type=ncV_AXIS, Channel=2, Disabled=TRUE, ModuleDisabled=FALSE)
  NcObject 8BVI0055HWD0.000-1_ncV_AXIS2 (ModuleId=8BVI0055HWD0.000-1_Zugband_Auslageband, Type=ncV_AXIS, Channel=2, Disabled=TRUE, ModuleDisabled=FALSE)
  NcObject 8B0P0440HW00.000-1_ncAXIS2 (ModuleId=8B0P0440HW00.000-1_Versorgung1, Type=ncAXIS, Channel=2, AcoposSimulation=Off, Disabled=TRUE, ModuleDisabled=FALSE)
  NcObject gMaster1 (ModuleId=8B0P0440HW00.000-1_Versorgung1, Type=ncV_AXIS, Channel=1, InitParameter=gmasteri, AdditionalData=PLCopen_ModPos="1000000,1", Disabled=FALSE, ModuleDisabled=FALSE)
  NcObject 8B0P0440HW00.000-1a_ncV_AXIS1 (ModuleId=8B0P0440HW00.000-1_Versorgung2, Type=ncV_AXIS, Channel=1, InitParameter=gmasteri, AdditionalData=PLCopen_ModPos="1000000,1", Disabled=FALSE, ModuleDisabled=FALSE)
  NcObject 8BVI0330HWSS.000-1_ncAXIS2 (ModuleId=8BVI0330HWSS.000-1_Stanzstation1, Type=ncAXIS, Channel=2, AcoposSimulation=Off, Disabled=TRUE, ModuleDisabled=FALSE)
  NcObject 8B0P0440HW00.000-1a_ncAXIS1 (ModuleId=8B0P0440HW00.000-1_Versorgung2, Type=ncAXIS, Channel=1, AcoposSimulation=Off, Disabled=TRUE, ModuleDisabled=FALSE)
  NcObject gUnwFeeder (ModuleId=8I64xxxxxxx.00x-1, ModuleAddress=SDC_IF1.ST1, Type=ncAXIS, Channel=1, AcoposSimulation=Off, InitParameter=gunwfeedi, AcoposParameter=gunwfeeda, AdditionalData=PLCopen_ModPos="118000,83" , Disabled=FALSE, ModuleDisabled=FALSE)
  NcObject gPackBelt (ModuleId=8I64xxxxxxx.00x-1a, ModuleAddress=SDC_IF1.ST2, Type=ncAXIS, Channel=1, AcoposSimulation=Off, InitParameter=gPackBelti, AcoposParameter=gPackBelta, AdditionalData=PLCopen_ModPos="118000,83" , Disabled=FALSE, ModuleDisabled=FALSE)
```

- Safety project (password-protected, skipped)

### Hardware.hw.as4
```
Module 0AC808.9 (Type=0AC808.9, Version=1.0.0.0)
  Connection (Connector=ETH1, TargetModule=5PC510.SX01-00, TargetConnector=IF3)
    Cable (Type=PowerlinkCable, Length=10, Version=1.0.0.3)
  Connection (Connector=ETH2, TargetModule=5PP520.1043-B50, TargetConnector=IF3)
    Cable (Type=PowerlinkCable, Length=10, Version=1.0.0.3)
  Connection (Connector=ETH3, TargetModule=5PP520.1043-B50a, TargetConnector=IF3)
    Cable (Type=PowerlinkCable, Length=10, Version=1.0.0.3)
Module 5AP920.1906-01 (Type=5AP920.1906-01, Version=2.1.0.0)
  VcObjectName = Visu
Module 5DLSDL.1000-01 (Type=5DLSDL.1000-01, Version=1.2.0.0)
  Connection (Connector=SDL1, TargetModule=5PP5IO.GMAC-00, TargetConnector=DS1)
  Connection (Connector=SL, TargetModule=5AP920.1906-01, TargetConnector=SL1)
Module 5PC510.SX01-00 (Type=5PC510.SX01-00, Version=2.1.5.0)
  Connector IF3:
    ActivateDevice = 1
    Mode = Manual
    InternetAddress = 192.168.1.10
    SubnetMask = 255.255.0.0
    InaNodeNumber = 0
    Vnc1
    VncVcObjectName1 = Visu
    VncKeyMappingFile1 = VC\PS2-Keyboard.dis
    VncAuthentication1 = 1
    VncPasswordViewOnly1 = v
    VncPasswordViewControl1 = c
Module 5PP520.1043-B50 (Type=5PP520.1043-B50, Version=2.0.1.2)
  Connection (Connector=IF3, TargetModule=0AC808.9, TargetConnector=ETH2, NodeNumber=64)
    Cable (Type=PowerlinkCable, Length=10, Version=1.0.0.3)
  Connector IF3 (NodeNumber=64)
  Terminal = true
  Mode = Manual
  InternetAddress = 192.168.1.64
  SubnetMask = 255.255.0.0
  VcObjectName = Visu1
Module 5PP520.1043-B50a (Type=5PP520.1043-B50, Version=2.0.1.2)
  Connection (Connector=IF3, TargetModule=0AC808.9, TargetConnector=ETH3, NodeNumber=65)
    Cable (Type=PowerlinkCable, Length=10, Version=1.0.0.3)
  Connector IF3 (NodeNumber=65)
  Terminal = true
  Mode = Manual
  InternetAddress = 192.168.1.65
  SubnetMask = 255.255.0.0
  VcObjectName = Visu2
Module 5PP5CP_US15_00 (Type=5PP5CP.US15-00, Version=2.1.6.0)
  Connection (Connector=SY, TargetModule=5PP520.1043-B50, TargetConnector=SY1)
  Terminal = true
  Temp.ProjectDirectory = C:\Users\s_spilker\Desktop\Spilker\projects\1_Actual\Nitto_26_07_18_2\
  Temp.ConfigurationName = Config1
Module 5PP5CP_US15_00a (Type=5PP5CP.US15-00, Version=2.1.6.0)
  Connection (Connector=SY, TargetModule=5PP520.1043-B50a, TargetConnector=SY1)
  Terminal = true
  Temp.ProjectDirectory = C:\Users\s_spilker\Desktop\Spilker\projects\1_Actual\Nitto_26_07_18_2\
  Temp.ConfigurationName = Config1
Module 5PP5CP_US15_02 (Type=5PP5CP.US15-02, Version=2.1.6.0)
  Connection (Connector=SY, TargetModule=5PC510.SX01-00, TargetConnector=SY1)
  UserRamDevice = PCI.1.PP5IF3.SRAM
  UserRamSize = 262144
  RemMemDevice = PCI.1.PP5IF3.SRAM
  RemMemSize = 131072
  PermanentPvSize = 16384
  RemanentGlobalPvSize = 98304
  PreservePermanentPvMemory = 1
  CyclicObjects = 200
  BRObjects = 350
  RebootReset = 1
  TimerDeviceType = EPLX2X
  TimerDevice = 5PP5IF.FPLM-00.IF1
  TaskClassIdleTime = 800
  Cyclic1Duration = 800
  Cyclic1Tolerance = 0
  Cyclic1Output = 1
  Cyclic2Duration = 2400
  Cyclic2Tolerance = 2400
  Cyclic3Duration = 10400
  Cyclic3Tolerance = 10400
  Cyclic8Duration = 8000
  FileDevice1
  FileDeviceName1 = USERPART
  FileDevicePath1 = F:\
Module 5PP5IF.FPLM-00 (Type=5PP5IF.FPLM-00, Version=2.5.0.0)
  Connection (Connector=SL, TargetModule=5PC510.SX01-00, TargetConnector=SL1)
  Connector IF1:
    DNAConfiguration = manual
    CycleTime = 800
Module 5PP5IO.GMAC-00 (Type=5PP5IO.GMAC-00, Version=2.2.2.0)
  Connection (Connector=SL, TargetModule=5PC510.SX01-00, TargetConnector=SL2)
Module 8B0P0440HW00.000-1_Versorgung1 (Type=8B0P0440HW00.000-1, Version=2.3.0.1)
  Connection (Connector=PLK1, TargetModule=X20HB2880, TargetConnector=ETH1, NodeNumber=4)
    Cable (Type=PowerlinkCable, Length=10, Version=1.0.0.3)
  Connection (Connector=PLK2, TargetModule=8B0P0440HW00.000-1_Versorgung2, TargetConnector=PLK1, NodeNumber=4)
    Cable (Type=PowerlinkCable, Length=10, Version=1.0.0.3)
Module 8B0P0440HW00.000-1_Versorgung2 (Type=8B0P0440HW00.000-1, Version=2.3.0.1)
  Connection (Connector=PLK1, TargetModule=8B0P0440HW00.000-1_Versorgung1, TargetConnector=PLK2, NodeNumber=5)
    Cable (Type=PowerlinkCable, Length=10, Version=1.0.0.3)
Module 8BAC0122.000-1 (Type=8BAC0122.000-1, Version=2.2.0.0)
  Connection (Connector=SS, TargetModule=8BVI0110HWD0.000-1_Hauptabrollung1und2, TargetConnector=SS2)
Module 8BAC0122.000-1a (Type=8BAC0122.000-1, Version=2.2.0.0)
  Connection (Connector=SS, TargetModule=8BVI0110HWD0.000-1_Hauptabrollung1und2, TargetConnector=SS1)
Module 8BAC0122.000-1b (Type=8BAC0122.000-1, Version=2.2.0.0)
  Connection (Connector=SS, TargetModule=8BVI0110HWD0.000-1_Bahnpuffer_Zugstation1, TargetConnector=SS1)
Module 8BAC0122.000-1c (Type=8BAC0122.000-1, Version=2.2.0.0)
  Connection (Connector=SS, TargetModule=8BVI0110HWD0.000-1_Bahnpuffer_Zugstation1, TargetConnector=SS2)
Module 8BAC0122.000-1d (Type=8BAC0122.000-1, Version=2.2.0.0)
  Connection (Connector=SS, TargetModule=8BVI0110HWD0.000-1_Gitteraufrollung1und2, TargetConnector=SS1)
Module 8BAC0122.000-1e (Type=8BAC0122.000-1, Version=2.2.0.0)
  Connection (Connector=SS, TargetModule=8BVI0110HWD0.000-1_Gitteraufrollung1und2, TargetConnector=SS2)
Module 8BAC0122.000-1f (Type=8BAC0122.000-1, Version=2.2.0.0)
  Connection (Connector=SS, TargetModule=8BVI0055HWD0.000-1_Zugband_Auslageband, TargetConnector=SS2)
Module 8BAC0122.000-1g (Type=8BAC0122.000-1, Version=2.2.0.0)
  Connection (Connector=SS, TargetModule=8BVI0055HWD0.000-1_Zugband_Auslageband, TargetConnector=SS1)
Module 8BAC0122.000-1h (Type=8BAC0122.000-1, Version=2.2.0.0)
  Connection (Connector=SS, TargetModule=8BVI0014HWD0.000-1_Fangband, TargetConnector=SS1)
Module 8BVI0014HWD0.000-1_Fangband (Type=8BVI0014HWD0.000-1, Version=2.3.0.1)
  Connection (Connector=PLK1, TargetModule=8BVI0014HWSS.000-1_Laengsschneider, TargetConnector=PLK2, NodeNumber=14)
    Cable (Type=PowerlinkCable, Length=10, Version=1.0.0.3)
  SupplyVoltage = 560
Module 8BVI0014HWSS.000-1_Laengsschneider (Type=8BVI0014HWSS.000-1, Version=2.3.0.1)
  Connection (Connector=PLK1, TargetModule=8BVI0055HWD0.000-1_Zugband_Auslageband, TargetConnector=PLK2, NodeNumber=13)
    Cable (Type=PowerlinkCable, Length=10, Version=1.0.0.3)
  Connection (Connector=PLK2, TargetModule=8BVI0014HWD0.000-1_Fangband, TargetConnector=PLK1, NodeNumber=13)
    Cable (Type=PowerlinkCable, Length=10, Version=1.0.0.3)
  SupplyVoltage = 560
Module 8BVI0055HWD0.000-1_Zugband_Auslageband (Type=8BVI0055HWD0.000-1, Version=2.3.0.1)
  Connection (Connector=PLK1, TargetModule=8BVI0110HWSS.000-1_GitterDrehfunktion, TargetConnector=PLK2, NodeNumber=12)
    Cable (Type=PowerlinkCable, Length=10, Version=1.0.0.3)
  Connection (Connector=PLK2, TargetModule=8BVI0014HWSS.000-1_Laengsschneider, TargetConnector=PLK1, NodeNumber=12)
    Cable (Type=PowerlinkCable, Length=10, Version=1.0.0.3)
  Connection (Connector=MT2, TargetModule=8LSA36.R0060D000-0, TargetConnector=MT)
  SupplyVoltage = 560
Module 8BVI0110HWD0.000-1_Bahnpuffer_Zugstation1 (Type=8BVI0110HWD0.000-1, Version=2.3.0.1)
  Connection (Connector=PLK1, TargetModule=8BVI0110HWD0.000-1_Hauptabrollung1und2, TargetConnector=PLK2, NodeNumber=9)
    Cable (Type=PowerlinkCable, Length=10, Version=1.0.0.3)
  Connection (Connector=PLK2, TargetModule=8BVI0110HWD0.000-1_Gitteraufrollung1und2, TargetConnector=PLK1, NodeNumber=9)
    Cable (Type=PowerlinkCable, Length=10, Version=1.0.0.3)
  Connection (Connector=MT2, TargetModule=8LSA46.R0045D000-0, TargetConnector=MT)
  SupplyVoltage = 560
Module 8BVI0110HWD0.000-1_Gitteraufrollung1und2 (Type=8BVI0110HWD0.000-1, Version=2.3.0.1)
  Connection (Connector=PLK1, TargetModule=8BVI0110HWD0.000-1_Bahnpuffer_Zugstation1, TargetConnector=PLK2, NodeNumber=10)
    Cable (Type=PowerlinkCable, Length=10, Version=1.0.0.3)
  Connection (Connector=PLK2, TargetModule=8BVI0110HWSS.000-1_GitterDrehfunktion, TargetConnector=PLK1, NodeNumber=10)
    Cable (Type=PowerlinkCable, Length=10, Version=1.0.0.3)
  Connection (Connector=MT2, TargetModule=8LSA55.R0045D100-1a, TargetConnector=MT)
  SupplyVoltage = 560
Module 8BVI0110HWD0.000-1_Hauptabrollung1und2 (Type=8BVI0110HWD0.000-1, Version=2.3.0.1)
  Connection (Connector=PLK1, TargetModule=8BVI0330HWSS.000-1_Stanzstation2, TargetConnector=PLK2, NodeNumber=8)
    Cable (Type=PowerlinkCable, Length=10, Version=1.0.0.3)
  Connection (Connector=PLK2, TargetModule=8BVI0110HWD0.000-1_Bahnpuffer_Zugstation1, TargetConnector=PLK1, NodeNumber=8)
    Cable (Type=PowerlinkCable, Length=10, Version=1.0.0.3)
  Connection (Connector=MT2, TargetModule=8LSN45.R0060D100-0, TargetConnector=MT)
  SupplyVoltage = 560
Module 8BVI0110HWSS.000-1_GitterDrehfunktion (Type=8BVI0110HWSS.000-1, Version=2.3.0.1)
  Connection (Connector=PLK1, TargetModule=8BVI0110HWD0.000-1_Gitteraufrollung1und2, TargetConnector=PLK2, NodeNumber=11)
    Cable (Type=PowerlinkCable, Length=10, Version=1.0.0.3)
  Connection (Connector=PLK2, TargetModule=8BVI0055HWD0.000-1_Zugband_Auslageband, TargetConnector=PLK1, NodeNumber=11)
    Cable (Type=PowerlinkCable, Length=10, Version=1.0.0.3)
  SupplyVoltage = 560
  FunctionModel = SingleAxis
Module 8BVI0330HWSS.000-1_Stanzstation1 (Type=8BVI0330HWSS.000-1, Version=2.3.0.1)
  Connection (Connector=PLK1, TargetModule=X20HB2880, TargetConnector=ETH2, NodeNumber=6)
    Cable (Type=PowerlinkCable, Length=10, Version=1.0.0.3)
  Connection (Connector=PLK2, TargetModule=8BVI0330HWSS.000-1_Stanzstation2, TargetConnector=PLK1, NodeNumber=6)
    Cable (Type=PowerlinkCable, Length=10, Version=1.0.0.3)
  SupplyVoltage = 560
Module 8BVI0330HWSS.000-1_Stanzstation2 (Type=8BVI0330HWSS.000-1, Version=2.3.0.1)
  Connection (Connector=PLK1, TargetModule=8BVI0330HWSS.000-1_Stanzstation1, TargetConnector=PLK2, NodeNumber=7)
    Cable (Type=PowerlinkCable, Length=10, Version=1.0.0.3)
  Connection (Connector=PLK2, TargetModule=8BVI0110HWD0.000-1_Hauptabrollung1und2, TargetConnector=PLK1, NodeNumber=7)
    Cable (Type=PowerlinkCable, Length=10, Version=1.0.0.3)
  SupplyVoltage = 560
Module 8BVSV2SAFE1-1 (Type=8BVSV2SAFE1-1, Version=1.10.3.1)
  Connection (Connector=SS, TargetModule=8BVI0330HWSS.000-1_Stanzstation1, TargetConnector=SS1)
  SafeModuleID = 5
Module 8BVSV2SAFE1-1a (Type=8BVSV2SAFE1-1, Version=1.10.3.1)
  Connection (Connector=SS, TargetModule=8BVI0330HWSS.000-1_Stanzstation2, TargetConnector=SS1)
  SafeModuleID = 6
Module 8BVSV2SAFE1-1b (Type=8BVSV2SAFE1-1, Version=1.10.3.1)
  Connection (Connector=SS, TargetModule=8BVI0110HWSS.000-1_GitterDrehfunktion, TargetConnector=SS1)
  SafeModuleID = 7
Module 8BVSV2SAFE1-1c (Type=8BVSV2SAFE1-1, Version=1.10.3.1)
  Connection (Connector=SS, TargetModule=8BVI0014HWSS.000-1_Laengsschneider, TargetConnector=SS1)
  SafeModuleID = 8
Module 8I64xxxxxxx.00x-1 (Type=8I64xxxxxxx.00x-1, Version=2.1.3.0)
  Connection (Connector=X2X1, TargetModule=X20BT9400_10A11, TargetConnector=X2X1)
    Cable (Type=X2XCable, Length=10, Version=1.0.0.3)
  Supervision = off
  ACC = 10
  DEC = 10
  HSP = 870
  ITH = 18
  UNS = 380
  NCR = 18
  NSP = 1380
  COS = 70
  TFR = 870
  COD = 0
  AxisIsPeriodic_r1 = on
Module 8I64xxxxxxx.00x-1a (Type=8I64xxxxxxx.00x-1, Version=2.1.3.0)
  Connection (Connector=X2X1, TargetModule=8I64xxxxxxx.00x-1, TargetConnector=X2X2)
    Cable (Type=X2XCable, Length=10, Version=1.0.0.3)
  Supervision = off
  HSP = 870
  ITH = 18
  UNS = 400
  NCR = 10
  NSP = 1420
  COS = 63
  TFR = 870
  COD = 0
  AxisIsPeriodic_r1 = on
Module 8LSA33.S0060D000-0 (Type=8LSA33.S0060D000-0, Version=1.0.1.34)
  Connection (Connector=EC, TargetModule=8BVSV2SAFE1-1c, TargetConnector=EC)
  Connection (Connector=MT, TargetModule=8BVI0014HWSS.000-1_Laengsschneider, TargetConnector=MT1)
Module 8LSA35.R2030D000-3 (Type=8LSA35.R2030D000-3, Version=2.2.0.0)
  Connection (Connector=EC, TargetModule=8BAC0122.000-1h, TargetConnector=EC)
  Connection (Connector=MT, TargetModule=8BVI0014HWD0.000-1_Fangband, TargetConnector=MT1)
Module 8LSA36.R0060D000-0 (Type=8LSA36.R0060D000-0, Version=1.0.1.40)
  Connection (Connector=EC, TargetModule=8BAC0122.000-1f, TargetConnector=EC)
  Connection (Connector=MT, TargetModule=8BVI0055HWD0.000-1_Zugband_Auslageband, TargetConnector=MT2)
Module 8LSA43.R0045D000-0 (Type=8LSA43.R0045D000-0, Version=1.0.1.40)
  Connection (Connector=EC, TargetModule=8BAC0122.000-1g, TargetConnector=EC)
  Connection (Connector=MT, TargetModule=8BVI0055HWD0.000-1_Zugband_Auslageband, TargetConnector=MT1)
Module 8LSA46.R0045D000-0 (Type=8LSA46.R0045D000-0, Version=1.0.1.40)
  Connection (Connector=EC, TargetModule=8BAC0122.000-1c, TargetConnector=EC)
  Connection (Connector=MT, TargetModule=8BVI0110HWD0.000-1_Bahnpuffer_Zugstation1, TargetConnector=MT2)
Module 8LSA55.R0045D100-1 (Type=8LSA55.R0045D100-1, Version=1.0.1.34)
  Connection (Connector=EC, TargetModule=8BAC0122.000-1d, TargetConnector=EC)
  Connection (Connector=MT, TargetModule=8BVI0110HWD0.000-1_Gitteraufrollung1und2, TargetConnector=MT1)
Module 8LSA55.R0045D100-1a (Type=8LSA55.R0045D100-1, Version=1.0.1.34)
  Connection (Connector=EC, TargetModule=8BAC0122.000-1e, TargetConnector=EC)
  Connection (Connector=MT, TargetModule=8BVI0110HWD0.000-1_Gitteraufrollung1und2, TargetConnector=MT2)
Module 8LSA55.R0045D200-1 (Type=8LSA55.R0045D200-1, Version=1.0.1.40)
  Connection (Connector=EC, TargetModule=8BAC0122.000-1b, TargetConnector=EC)
  Connection (Connector=MT, TargetModule=8BVI0110HWD0.000-1_Bahnpuffer_Zugstation1, TargetConnector=MT1)
Module 8LSA55.S0045D300-1 (Type=8LSA55.S0045D300-1, Version=1.0.1.34)
  Connection (Connector=EC, TargetModule=8BVSV2SAFE1-1b, TargetConnector=EC)
  Connection (Connector=MT, TargetModule=8BVI0110HWSS.000-1_GitterDrehfunktion, TargetConnector=MT1)
Module 8LSA75.S0030D000-0 (Type=8LSA75.S0030D000-0, Version=1.0.1.34)
  Connection (Connector=EC, TargetModule=8BVSV2SAFE1-1, TargetConnector=EC)
  Connection (Connector=MT, TargetModule=8BVI0330HWSS.000-1_Stanzstation1, TargetConnector=MT1)
Module 8LSA75.S0030D000-0a (Type=8LSA75.S0030D000-0, Version=1.0.1.34)
  Connection (Connector=EC, TargetModule=8BVSV2SAFE1-1a, TargetConnector=EC)
  Connection (Connector=MT, TargetModule=8BVI0330HWSS.000-1_Stanzstation2, TargetConnector=MT1)
Module 8LSN45.R0060D100-0 (Type=8LSN45.R0060D100-0, Version=1.0.1.34)
  Connection (Connector=EC, TargetModule=8BAC0122.000-1, TargetConnector=EC)
  Connection (Connector=MT, TargetModule=8BVI0110HWD0.000-1_Hauptabrollung1und2, TargetConnector=MT2)
Module 8LSN45.R0060D100-0a (Type=8LSN45.R0060D100-0, Version=1.0.1.34)
  Connection (Connector=EC, TargetModule=8BAC0122.000-1a, TargetConnector=EC)
  Connection (Connector=MT, TargetModule=8BVI0110HWD0.000-1_Hauptabrollung1und2, TargetConnector=MT1)
Module X20AI1744_101A6 (Type=X20AI1744, Version=1.10.0.0)
  Connection (Connector=SS1, TargetModule=X20TB12af, TargetConnector=SS)
  Connection (Connector=SL, TargetModule=X20BM11ad, TargetConnector=SL1)
Module X20AI4622_101A5 (Type=X20AI4622, Version=1.2.0.0)
  Connection (Connector=SS1, TargetModule=X20TB12h, TargetConnector=SS)
  Connection (Connector=SL, TargetModule=X20BM11ab, TargetConnector=SL1)
  Supervision = off
  ChannelType01 = 4 to 20mA
Module X20AI4622_10A12 (Type=X20AI4622, Version=1.2.0.0)
  Connection (Connector=SS1, TargetModule=X20TB12ae, TargetConnector=SS)
  Connection (Connector=SL, TargetModule=X20BM11ac, TargetConnector=SL1)
  Supervision = off
Module X20AI4622_202A8 (Type=X20AI4622, Version=1.2.0.0)
  Connection (Connector=SS1, TargetModule=X20TB12aa, TargetConnector=SS)
  Connection (Connector=SL, TargetModule=X20BM11x, TargetConnector=SL1)
Module X20BB80_101A1 (Type=X20BB80, Version=1.1.0.0)
  Connector IF1:
    CycleTime = 800
Module X20BB80_201A1 (Type=X20BB80, Version=1.1.0.0)
  Connector IF1:
    CycleTime = 800
Module X20BB82_9A2 (Type=X20BB82, Version=1.1.0.0)
  Connector IF1:
    CycleTime = 800
Module X20BC0083 (Type=X20BC0083, Version=2.14.0.0)
  Connection (Connector=PLK1, TargetModule=X20BC8083, TargetConnector=PLK2, NodeNumber=15)
    Cable (Type=PowerlinkCable, Length=10, Version=1.0.0.3)
  Connection (Connector=PLK2, TargetModule=X20BC0083a, TargetConnector=PLK1, NodeNumber=15)
    Cable (Type=PowerlinkCable, Length=10, Version=1.0.0.3)
  Connection (Connector=SL, TargetModule=X20BB80_101A1, TargetConnector=SL1)
Module X20BC0083a (Type=X20BC0083, Version=2.14.0.0)
  Connection (Connector=PLK1, TargetModule=X20BC0083, TargetConnector=PLK2, NodeNumber=16)
    Cable (Type=PowerlinkCable, Length=10, Version=1.0.0.3)
  Connection (Connector=SL, TargetModule=X20BB80_201A1, TargetConnector=SL1)
Module X20BC8083 (Type=X20BC8083, Version=2.14.0.0)
  Connection (Connector=PLK1, TargetModule=X20SL8010_9A1, TargetConnector=PLK2, NodeNumber=3)
    Cable (Type=PowerlinkCable, Length=10, Version=1.0.0.3)
  Connection (Connector=PLK2, TargetModule=X20BC0083, TargetConnector=PLK1, NodeNumber=3)
    Cable (Type=PowerlinkCable, Length=10, Version=1.0.0.3)
  Connection (Connector=SL, TargetModule=X20BB82_9A2, TargetConnector=SL1)
Module X20BM11 (Type=X20BM11, Version=1.1.0.0)
  Connection (Connector=X2X1, TargetModule=X20BM11f, TargetConnector=X2X2)
Module X20BM11a (Type=X20BM11, Version=1.1.0.0)
  Connection (Connector=X2X1, TargetModule=X20BM11, TargetConnector=X2X2)
Module X20BM11aa (Type=X20BM11, Version=1.1.0.0)
  Connection (Connector=X2X1, TargetModule=X20BM11z, TargetConnector=X2X2)
Module X20BM11ab (Type=X20BM11, Version=1.1.0.0)
  Connection (Connector=X2X1, TargetModule=X20BM33d, TargetConnector=X2X2)
Module X20BM11ac (Type=X20BM11, Version=1.1.0.0)
  Connection (Connector=X2X1, TargetModule=X20BM11e, TargetConnector=X2X2)
Module X20BM11ad (Type=X20BM11, Version=1.1.0.0)
  Connection (Connector=X2X1, TargetModule=X20BM11ab, TargetConnector=X2X2)
Module X20BM11b (Type=X20BM11, Version=1.1.0.0)
  Connection (Connector=X2X1, TargetModule=X20BM11a, TargetConnector=X2X2)
Module X20BM11c (Type=X20BM11, Version=1.1.0.0)
  Connection (Connector=X2X1, TargetModule=X20BM11b, TargetConnector=X2X2)
Module X20BM11d (Type=X20BM11, Version=1.1.0.0)
  Connection (Connector=X2X1, TargetModule=X20BM11c, TargetConnector=X2X2)
Module X20BM11e (Type=X20BM11, Version=1.1.0.0)
  Connection (Connector=X2X1, TargetModule=X20BM11d, TargetConnector=X2X2)
Module X20BM11f (Type=X20BM11, Version=1.1.0.0)
  Connection (Connector=X2X1, TargetModule=X20BM33f, TargetConnector=X2X2)
Module X20BM11g (Type=X20BM11, Version=1.1.0.0)
  Connection (Connector=X2X1, TargetModule=X20BM11ac, TargetConnector=X2X2)
Module X20BM11h (Type=X20BM11, Version=1.1.0.0)
  Connection (Connector=X2X1, TargetModule=X20BB80_101A1, TargetConnector=IF1)
Module X20BM11i (Type=X20BM11, Version=1.1.0.0)
  Connection (Connector=X2X1, TargetModule=X20BM11ad, TargetConnector=X2X2)
Module X20BM11j (Type=X20BM11, Version=1.1.0.0)
  Connection (Connector=X2X1, TargetModule=X20BM11i, TargetConnector=X2X2)
Module X20BM11k (Type=X20BM11, Version=1.1.0.0)
  Connection (Connector=X2X1, TargetModule=X20BM11j, TargetConnector=X2X2)
Module X20BM11l (Type=X20BM11, Version=1.1.0.0)
  Connection (Connector=X2X1, TargetModule=X20BM11k, TargetConnector=X2X2)
Module X20BM11m (Type=X20BM11, Version=1.1.0.0)
  Connection (Connector=X2X1, TargetModule=X20BM11l, TargetConnector=X2X2)
Module X20BM11n (Type=X20BM11, Version=1.1.0.0)
  Connection (Connector=X2X1, TargetModule=X20BM11m, TargetConnector=X2X2)
Module X20BM11o (Type=X20BM11, Version=1.1.0.0)
  Connection (Connector=X2X1, TargetModule=X20BM11n, TargetConnector=X2X2)
Module X20BM11p (Type=X20BM11, Version=1.1.0.0)
  Connection (Connector=X2X1, TargetModule=X20BM11o, TargetConnector=X2X2)
Module X20BM11q (Type=X20BM11, Version=1.1.0.0)
  Connection (Connector=X2X1, TargetModule=X20BM33g, TargetConnector=X2X2)
Module X20BM11r (Type=X20BM11, Version=1.1.0.0)
  Connection (Connector=X2X1, TargetModule=X20BM11q, TargetConnector=X2X2)
Module X20BM11s (Type=X20BM11, Version=1.1.0.0)
  Connection (Connector=X2X1, TargetModule=X20BM11r, TargetConnector=X2X2)
Module X20BM11t (Type=X20BM11, Version=1.1.0.0)
  Connection (Connector=X2X1, TargetModule=X20BM11s, TargetConnector=X2X2)
Module X20BM11u (Type=X20BM11, Version=1.1.0.0)
  Connection (Connector=X2X1, TargetModule=X20BM11t, TargetConnector=X2X2)
Module X20BM11v (Type=X20BM11, Version=1.1.0.0)
  Connection (Connector=X2X1, TargetModule=X20BM11u, TargetConnector=X2X2)
Module X20BM11w (Type=X20BM11, Version=1.1.0.0)
  Connection (Connector=X2X1, TargetModule=X20BM11v, TargetConnector=X2X2)
Module X20BM11x (Type=X20BM11, Version=1.1.0.0)
  Connection (Connector=X2X1, TargetModule=X20BM11w, TargetConnector=X2X2)
Module X20BM11y (Type=X20BM11, Version=1.1.0.0)
  Connection (Connector=X2X1, TargetModule=X20BM11x, TargetConnector=X2X2)
Module X20BM11z (Type=X20BM11, Version=1.1.0.0)
  Connection (Connector=X2X1, TargetModule=X20BM11y, TargetConnector=X2X2)
Module X20BM33 (Type=X20BM33, Version=1.1.0.0)
  Connection (Connector=X2X1, TargetModule=X20BB82_9A2, TargetConnector=IF1)
Module X20BM33a (Type=X20BM33, Version=1.1.0.0)
  Connection (Connector=X2X1, TargetModule=X20BM33, TargetConnector=X2X2)
Module X20BM33b (Type=X20BM33, Version=1.1.0.0)
  Connection (Connector=X2X1, TargetModule=X20BM33a, TargetConnector=X2X2)
Module X20BM33c (Type=X20BM33, Version=1.1.0.0)
  Connection (Connector=X2X1, TargetModule=X20BM11h, TargetConnector=X2X2)
Module X20BM33d (Type=X20BM33, Version=1.1.0.0)
  Connection (Connector=X2X1, TargetModule=X20BM33c, TargetConnector=X2X2)
Module X20BM33e (Type=X20BM33, Version=1.1.0.0)
  Connection (Connector=X2X1, TargetModule=X20BB80_201A1, TargetConnector=IF1)
Module X20BM33f (Type=X20BM33, Version=1.1.0.0)
  Connection (Connector=X2X1, TargetModule=X20BM33b, TargetConnector=X2X2)
Module X20BM33g (Type=X20BM33, Version=1.1.0.0)
  Connection (Connector=X2X1, TargetModule=X20BM33e, TargetConnector=X2X2)
Module X20BT9400_10A11 (Type=X20BT9400, Version=1.3.0.0)
  Connection (Connector=SL, TargetModule=X20BM11g, TargetConnector=SL1)
  Supervision = off
Module X20DC1196_202A9 (Type=X20DC1196, Version=1.4.0.0)
  Connection (Connector=SS1, TargetModule=X20TB12ab, TargetConnector=SS)
  Connection (Connector=SL, TargetModule=X20BM11y, TargetConnector=SL1)
Module X20DI9371_102A2 (Type=X20DI9371, Version=1.4.0.0)
  Connection (Connector=SS1, TargetModule=X20TB12m, TargetConnector=SS)
  Connection (Connector=SL, TargetModule=X20BM11j, TargetConnector=SL1)
Module X20DI9371_102A3 (Type=X20DI9371, Version=1.4.0.0)
  Connection (Connector=SS1, TargetModule=X20TB12n, TargetConnector=SS)
  Connection (Connector=SL, TargetModule=X20BM11k, TargetConnector=SL1)
Module X20DI9371_102A4 (Type=X20DI9371, Version=1.4.0.0)
  Connection (Connector=SS1, TargetModule=X20TB12o, TargetConnector=SS)
  Connection (Connector=SL, TargetModule=X20BM11l, TargetConnector=SL1)
Module X20DI9371_10A5 (Type=X20DI9371, Version=1.4.0.0)
  Connection (Connector=SS1, TargetModule=X20TB12a, TargetConnector=SS)
  Connection (Connector=SL, TargetModule=X20BM11, TargetConnector=SL1)
  Supervision = off
Module X20DI9371_10A6 (Type=X20DI9371, Version=1.4.0.0)
  Connection (Connector=SS1, TargetModule=X20TB12b, TargetConnector=SS)
  Connection (Connector=SL, TargetModule=X20BM11a, TargetConnector=SL1)
  Supervision = off
Module X20DI9371_10A7 (Type=X20DI9371, Version=1.4.0.0)
  Connection (Connector=SS1, TargetModule=X20TB12c, TargetConnector=SS)
  Connection (Connector=SL, TargetModule=X20BM11b, TargetConnector=SL1)
  Supervision = off
Module X20DI9371_202A2 (Type=X20DI9371, Version=1.4.0.0)
  Connection (Connector=SS1, TargetModule=X20TB12u, TargetConnector=SS)
  Connection (Connector=SL, TargetModule=X20BM11r, TargetConnector=SL1)
Module X20DI9371_202A3 (Type=X20DI9371, Version=1.4.0.0)
  Connection (Connector=SS1, TargetModule=X20TB12v, TargetConnector=SS)
  Connection (Connector=SL, TargetModule=X20BM11s, TargetConnector=SL1)
Module X20DI9371_202A4 (Type=X20DI9371, Version=1.4.0.0)
  Connection (Connector=SS1, TargetModule=X20TB12w, TargetConnector=SS)
  Connection (Connector=SL, TargetModule=X20BM11t, TargetConnector=SL1)
Module X20DI9371_202A5 (Type=X20DI9371, Version=1.4.0.0)
  Connection (Connector=SS1, TargetModule=X20TB12x, TargetConnector=SS)
  Connection (Connector=SL, TargetModule=X20BM11u, TargetConnector=SL1)
Module X20DO4332_102A8 (Type=X20DO4332, Version=1.6.0.0)
  Connection (Connector=SS1, TargetModule=X20TB12s, TargetConnector=SS)
  Connection (Connector=SL, TargetModule=X20BM11p, TargetConnector=SL1)
  Supervision = off
Module X20DO9322_102A5 (Type=X20DO9322, Version=1.5.0.0)
  Connection (Connector=SS1, TargetModule=X20TB12p, TargetConnector=SS)
  Connection (Connector=SL, TargetModule=X20BM11m, TargetConnector=SL1)
Module X20DO9322_102A6 (Type=X20DO9322, Version=1.5.0.0)
  Connection (Connector=SS1, TargetModule=X20TB12q, TargetConnector=SS)
  Connection (Connector=SL, TargetModule=X20BM11n, TargetConnector=SL1)
Module X20DO9322_10A10 (Type=X20DO9322, Version=1.5.0.0)
  Connection (Connector=SS1, TargetModule=X20TB12f, TargetConnector=SS)
  Connection (Connector=SL, TargetModule=X20BM11e, TargetConnector=SL1)
  Supervision = off
Module X20DO9322_10A8 (Type=X20DO9322, Version=1.5.0.0)
  Connection (Connector=SS1, TargetModule=X20TB12d, TargetConnector=SS)
  Connection (Connector=SL, TargetModule=X20BM11c, TargetConnector=SL1)
  Supervision = off
Module X20DO9322_10A9 (Type=X20DO9322, Version=1.5.0.0)
  Connection (Connector=SS1, TargetModule=X20TB12e, TargetConnector=SS)
  Connection (Connector=SL, TargetModule=X20BM11d, TargetConnector=SL1)
  Supervision = off
Module X20DO9322_202A11 (Type=X20DO9322, Version=1.5.0.0)
  Connection (Connector=SS1, TargetModule=X20TB12ad, TargetConnector=SS)
  Connection (Connector=SL, TargetModule=X20BM11aa, TargetConnector=SL1)
  Supervision = off
Module X20DO9322_202A6 (Type=X20DO9322, Version=1.5.0.0)
  Connection (Connector=SS1, TargetModule=X20TB12y, TargetConnector=SS)
  Connection (Connector=SL, TargetModule=X20BM11v, TargetConnector=SL1)
Module X20DO9322_202A7 (Type=X20DO9322, Version=1.5.0.0)
  Connection (Connector=SS1, TargetModule=X20TB12z, TargetConnector=SS)
  Connection (Connector=SL, TargetModule=X20BM11w, TargetConnector=SL1)
Module X20DS4387_101A2 (Type=X20DS4387, Version=1.3.0.0)
  Connection (Connector=SS1, TargetModule=X20TB12k, TargetConnector=SS)
  Connection (Connector=SL, TargetModule=X20BM11h, TargetConnector=SL1)
  DataSizeOut01 = 2
  Mode02 = Operate
  DataSizeOut02 = 3
Module X20HB2880 (Type=X20HB2880, Version=1.2.0.0)
  Connection (Connector=ETH1, TargetModule=8B0P0440HW00.000-1_Versorgung1, TargetConnector=PLK1)
    Cable (Type=PowerlinkCable, Length=10, Version=1.0.0.3)
  Connection (Connector=ETH2, TargetModule=8BVI0330HWSS.000-1_Stanzstation1, TargetConnector=PLK1)
    Cable (Type=PowerlinkCable, Length=10, Version=1.0.0.3)
  Connection (Connector=SS, TargetModule=X20BB82_9A2, TargetConnector=SS1)
Module X20MK0201 (Type=X20MK0201, Version=1.0.0.0)
  Connection (Connector=SL, TargetModule=X20SL8010_9A1, TargetConnector=SL1)
Module X20PS2100_102A7 (Type=X20PS2100, Version=1.4.0.0)
  Connection (Connector=SS1, TargetModule=X20TB12r, TargetConnector=SS)
  Connection (Connector=SL, TargetModule=X20BM11o, TargetConnector=SL1)
  Supervision = off
Module X20PS2100_202A10 (Type=X20PS2100, Version=1.4.0.0)
  Connection (Connector=SS1, TargetModule=X20TB12ac, TargetConnector=SS)
  Connection (Connector=SL, TargetModule=X20BM11z, TargetConnector=SL1)
  Supervision = off
Module X20PS3300_102A1 (Type=X20PS3300, Version=1.4.0.0)
  Connection (Connector=SS1, TargetModule=X20TB12l, TargetConnector=SS)
  Connection (Connector=SL, TargetModule=X20BM11i, TargetConnector=SL1)
Module X20PS3300_10A4 (Type=X20PS3300, Version=1.4.0.0)
  Connection (Connector=SS1, TargetModule=X20TB12g, TargetConnector=SS)
  Connection (Connector=SL, TargetModule=X20BM11f, TargetConnector=SL1)
  Supervision = off
Module X20PS3300_202A1 (Type=X20PS3300, Version=1.4.0.0)
  Connection (Connector=SS1, TargetModule=X20TB12t, TargetConnector=SS)
  Connection (Connector=SL, TargetModule=X20BM11q, TargetConnector=SL1)
Module X20PS9400 (Type=X20PS9400, Version=1.8.0.0)
  Connection (Connector=SS1, TargetModule=X20TB12, TargetConnector=SS)
  Connection (Connector=PS, TargetModule=X20BB82_9A2, TargetConnector=PS1)
Module X20PS9400a (Type=X20PS9400, Version=1.8.0.0)
  Connection (Connector=SS1, TargetModule=X20TB12i, TargetConnector=SS)
  Connection (Connector=PS, TargetModule=X20BB80_101A1, TargetConnector=PS1)
Module X20PS9400b (Type=X20PS9400, Version=1.8.0.0)
  Connection (Connector=SS1, TargetModule=X20TB12j, TargetConnector=SS)
  Connection (Connector=PS, TargetModule=X20BB80_201A1, TargetConnector=PS1)
Module X20SI4100_10A1 (Type=X20SI4100, Version=1.10.12.0)
  Connection (Connector=SS1, TargetModule=X20TB52a, TargetConnector=SS)
  Connection (Connector=SL, TargetModule=X20BM33, TargetConnector=SL1)
  Supervision = off
Module X20SI4100_10A2 (Type=X20SI4100, Version=1.10.12.0)
  Connection (Connector=SS1, TargetModule=X20TB52b, TargetConnector=SS)
  Connection (Connector=SL, TargetModule=X20BM33a, TargetConnector=SL1)
  Supervision = off
  SafeModuleID = 3
Module X20SI4100_201A3 (Type=X20SI4100, Version=1.10.12.0)
  Connection (Connector=SS1, TargetModule=X20TB52k, TargetConnector=SS)
  Connection (Connector=SL, TargetModule=X20BM33g, TargetConnector=SL1)
  Supervision = off
  SafeModuleID = 13
Module X20SI9100_101A3 (Type=X20SI9100, Version=1.10.12.0)
  Connection (Connector=SS1, TargetModule=X20TB52d, TargetConnector=SS)
  Connection (Connector=SS2, TargetModule=X20TB52e, TargetConnector=SS)
  Connection (Connector=SL, TargetModule=X20BM33c, TargetConnector=SL1)
  Supervision = off
  SafeModuleID = 9
Module X20SI9100_101A4 (Type=X20SI9100, Version=1.10.12.0)
  Connection (Connector=SS1, TargetModule=X20TB52f, TargetConnector=SS)
  Connection (Connector=SS2, TargetModule=X20TB52g, TargetConnector=SS)
  Connection (Connector=SL, TargetModule=X20BM33d, TargetConnector=SL1)
  Supervision = off
  SafeModuleID = 10
Module X20SI9100_201A2 (Type=X20SI9100, Version=1.10.12.0)
  Connection (Connector=SS1, TargetModule=X20TB52h, TargetConnector=SS)
  Connection (Connector=SS2, TargetModule=X20TB52i, TargetConnector=SS)
  Connection (Connector=SL, TargetModule=X20BM33e, TargetConnector=SL1)
  Supervision = off
  SafeModuleID = 11
Module X20SL8010_9A1 (Type=X20SL8010, Version=1.6.5.2)
  Connection (Connector=PLK1, TargetModule=5PP5IF.FPLM-00, TargetConnector=IF1, NodeNumber=2)
    Cable (Type=PowerlinkCable, Length=10, Version=1.0.0.3)
  Connection (Connector=PLK2, TargetModule=X20BC8083, TargetConnector=PLK1, NodeNumber=2)
    Cable (Type=PowerlinkCable, Length=10, Version=1.0.0.3)
  Connection (Connector=SS1, TargetModule=X20TB52, TargetConnector=SS)
  Supervision = off
  SafeProject = SafeDESIGNER Projekt
  SafeDesigner = 2.90.21.261733
Module X20SO4110_10A13 (Type=X20SO4110, Version=1.10.12.0)
  Connection (Connector=SS1, TargetModule=X20TB52j, TargetConnector=SS)
  Connection (Connector=SL, TargetModule=X20BM33f, TargetConnector=SL1)
  Supervision = off
  SafeModuleID = 12
  MaxSwitchFreq_01 = 10Hz
  DigitalOutput01 = viaSafeLOGIC
Module X20SO4110_10A3 (Type=X20SO4110, Version=1.10.12.0)
  Connection (Connector=SS1, TargetModule=X20TB52c, TargetConnector=SS)
  Connection (Connector=SL, TargetModule=X20BM33b, TargetConnector=SL1)
  Supervision = off
  SafeModuleID = 4
  DigitalOutput01 = viaSafeLOGIC
  DigitalOutput02 = viaSafeLOGIC
  DigitalOutput03 = viaSafeLOGIC
  DigitalOutput04 = viaSafeLOGIC
Module X20TB12 (Type=X20TB12, Version=1.0.0.0)
Module X20TB12a (Type=X20TB12, Version=1.0.0.0)
Module X20TB12aa (Type=X20TB12, Version=1.0.0.0)
Module X20TB12ab (Type=X20TB12, Version=1.0.0.0)
Module X20TB12ac (Type=X20TB12, Version=1.0.0.0)
Module X20TB12ad (Type=X20TB12, Version=1.0.0.0)
Module X20TB12ae (Type=X20TB12, Version=1.0.0.0)
Module X20TB12af (Type=X20TB12, Version=1.0.0.0)
Module X20TB12b (Type=X20TB12, Version=1.0.0.0)
Module X20TB12c (Type=X20TB12, Version=1.0.0.0)
Module X20TB12d (Type=X20TB12, Version=1.0.0.0)
Module X20TB12e (Type=X20TB12, Version=1.0.0.0)
Module X20TB12f (Type=X20TB12, Version=1.0.0.0)
Module X20TB12g (Type=X20TB12, Version=1.0.0.0)
Module X20TB12h (Type=X20TB12, Version=1.0.0.0)
Module X20TB12i (Type=X20TB12, Version=1.0.0.0)
Module X20TB12j (Type=X20TB12, Version=1.0.0.0)
Module X20TB12k (Type=X20TB12, Version=1.0.0.0)
Module X20TB12l (Type=X20TB12, Version=1.0.0.0)
Module X20TB12m (Type=X20TB12, Version=1.0.0.0)
Module X20TB12n (Type=X20TB12, Version=1.0.0.0)
Module X20TB12o (Type=X20TB12, Version=1.0.0.0)
Module X20TB12p (Type=X20TB12, Version=1.0.0.0)
Module X20TB12q (Type=X20TB12, Version=1.0.0.0)
Module X20TB12r (Type=X20TB12, Version=1.0.0.0)
Module X20TB12s (Type=X20TB12, Version=1.0.0.0)
Module X20TB12t (Type=X20TB12, Version=1.0.0.0)
Module X20TB12u (Type=X20TB12, Version=1.0.0.0)
Module X20TB12v (Type=X20TB12, Version=1.0.0.0)
Module X20TB12w (Type=X20TB12, Version=1.0.0.0)
Module X20TB12x (Type=X20TB12, Version=1.0.0.0)
Module X20TB12y (Type=X20TB12, Version=1.0.0.0)
Module X20TB12z (Type=X20TB12, Version=1.0.0.0)
Module X20TB52 (Type=X20TB52, Version=1.0.0.2)
Module X20TB52a (Type=X20TB52, Version=1.0.0.2)
Module X20TB52b (Type=X20TB52, Version=1.0.0.2)
Module X20TB52c (Type=X20TB52, Version=1.0.0.2)
Module X20TB52d (Type=X20TB52, Version=1.0.0.2)
Module X20TB52e (Type=X20TB52, Version=1.0.0.2)
Module X20TB52f (Type=X20TB52, Version=1.0.0.2)
Module X20TB52g (Type=X20TB52, Version=1.0.0.2)
Module X20TB52h (Type=X20TB52, Version=1.0.0.2)
Module X20TB52i (Type=X20TB52, Version=1.0.0.2)
Module X20TB52j (Type=X20TB52, Version=1.0.0.2)
Module X20TB52k (Type=X20TB52, Version=1.0.0.2)
```

## Configuration Simulation

CPU , AutomationRuntime V4.04, Build 4.1.2, Safety 0.0

### Task classes (Cpu.sw)
```
Cyclic#2:
  MAIN <- MainMachineCtrl.MAIN.prg
Cyclic#3:
  csv_hdl <- pkgRecipe.csv_hdl.prg
  tool_hdl <- pkgRecipe.tool_hdl.prg
  al_hdl <- pkgRecipe.al_hdl.prg
  picctrl <- pkgRecipe.picctrl.prg
  save2USB <- pkgRecipe.save2USB.prg
  VisuRange <- Visualization.VisuCycl.VisuRange.prg
  VisuPages <- Visualization.VisuCycl.VisuPages.prg
  VisuTasks <- Visualization.VisuCycl.VisuTasks.prg
DataObjects: Acp10sys
VcDataObjects: Visu <- Visualization.VisuCycl.Visu.dob
Binaries: iomap, asfw, sysconf, arconfig, ashwd, acp10map, acp10cfg, vccovl, visvc, vcfntttf, vccpopup, vccshape, vcctext, vccddbox, arial, vctcal, vccdt, vccbtn, vccnum, vcpfar00, vcdsint, Visu02, vcpdvnc, vcpdsw, vcalarm, vcchspot, vcfile, vcmgr, vccstr, vcresman, vcgclass, vcdsloc, arialbd, vcnet, Visu03, vcrt, vccalarm, vcclbox, vccbmp, vcbclass, vcshared, vccline, Visu01
Libraries: AsWndCon, CSV_File, HlpStr, AsTime, AsBrMath, AsBrStr, AsMem, FileIO, UserVC, UserSpilke, Acp10man, Bibliothek, Acp10par, NcGlobal, Acp10_MC, AsMath, SprRegMa, SprGeneral, TorqueCtrl, LoopConR, runtime, asstring, standard, sys_lib, asieccon, visapi, brsystem, powerlnk, asusb, dataobj
```

### Hardware.hw.as4
```
Module PC_any (Type=PC_any, Version=1.1.0.0, OrderNumber=PC)
  Connector IF3:
    Vnc1
    VncVcObjectName1 = Visu
    VncAuthentication1 = 1
    VncPasswordViewOnly1 = v
    VncPasswordViewControl1 = c
    VncRefreshRate1 = 200
  PermanentPvSize = 4096
  Cyclic1Duration = 100000
  Cyclic1Tolerance = 10000000
  Cyclic2Duration = 100000
  Cyclic2Tolerance = 10000000
  Cyclic3Duration = 100000
  Cyclic3Tolerance = 10000000
  Cyclic4Duration = 1000000
  Cyclic4Tolerance = 10000000
  Cyclic5Duration = 2000000
  Cyclic5Tolerance = 10000000
  Cyclic6Duration = 3000000
  Cyclic6Tolerance = 12000000
  Cyclic7Duration = 4000000
  Cyclic7Tolerance = 12000000
  Cyclic8Duration = 5000000
  Cyclic8Tolerance = 30000000
```

### Cpu.per - PC_any/Cpu.per
```iecst
(********************************************************************
 * COPYRIGHT --
 ********************************************************************
 * Datei: Cpu.per
 * Autor: sbueker
 * Erstellt: 15. Juli 2014
 ********************************************************************
 * Deklaration der permanenten Variablen
 ********************************************************************)
VAR_CONFIG
	gMachRecipe AT %M0; (* *)
	gApplRecipe AT %M432; (* *)
END_VAR
```

### Acp10cfg.ncc - PC_any/Motion/Acp10cfg.ncc
```
NcConfiguration (Version=2.37.0, NcSwId=Acp10)
  ACP10CF1_typ:
    cnt_nettrc_rec_drive = 150
    bufsize_trace_upload = 1200
    tc_nc_man_task = Cyclic #1
    glob_pv_as_ncobject = Yes
    ncsys_dl_broadcast = Yes
    ncsys_dl_acp_reset = Yes
    network_init:
      ncsw_init_execute = Yes
      automatic_execute = No
      node_nr_warning = Yes
      net_err_before_ncact = Yes
    nettrc:
      enter_parsecrec = Yes
      enter_ncaction = Yes
      save_ring_startidx = No
```

## Logical view

Binary libraries used (declarations not repeated): operator, runtime, astime, AsIecCon, Acp10man 2.37.0, Acp10par 2.37.0, NcGlobal 2.37.0, AsARCfg, AsBrMath, AsBrStr, AsMem, asstring, AsUSB, brsystem, FileIO, LoopConR 2.80.2, powerlnk, standard, sys_lib, Visapi, Acp10_MC 2.37.0, Acp10sdc 2.37.0, SafeMC 2.37.0, MC_RegMa 2.37.0, AsMath, Acp10sim 2.37.0, AsWndCon 1.11.6

### Package Logical/Documentation - Paket

- Antrieb_Berechnungen_NITTO.xlsx (binary file, 59051 bytes)
### Global.var - Globale Variablen
```iecst
(********************************************************************
 * COPYRIGHT -- Microsoft
 ********************************************************************
 * Datei: Global.var
 * Autor: okrebs
 * Erstellt: 22. Mai 2014
 ********************************************************************
 * Globale Variablen des Projekts Nitto_40
 ********************************************************************)
(*Global Machine structure*)
VAR
	gNewOutputBrake : BOOL;
	gMachine : Machine_Type;
	CONST : FB_CONST_MASCHINE;
END_VAR
VAR RETAIN
	gPaperCounter : UDINT;
	gProductCounter : UDINT; (*total amount of produced products*)
	gMeterCounter : UDINT; (*total travelled distance of master axis [0.01m]*)
	gMeterCounterTotal : UDINT; (*total travelled distance of master axis [0.01m]*)
	gMachRecipe : rcp_machine_typ;
	gApplRecipe : rcp_prog_typ;
	gCuttinRecipe : rcp_cutting_typ;
	gPermValid : UDINT;
	gWinderRecipeData : FB_WinderRecipeData; (*TODO: Bitte Kommentar hier einzufügen*)
END_VAR
(*Variables from Visu*)
VAR
	gVisu : Visu_Type;
END_VAR
(*Drive variables and constants*)
VAR
	gUnwinder : ACP10AXIS_typ;
	gMaster1 : ACP10AXIS_typ; (*Virtueller Master*)
	gCut1 : ACP10AXIS_typ; (*Stanzstation 1*)
	gCut2 : ACP10AXIS_typ; (*Stanzstation 2*)
	gGridLeft : ACP10AXIS_typ; (*Gitteraufwickler 1*)
	gGridRight : ACP10AXIS_typ; (*Gitteraufwickler 2*)
	gPBS1 : ACP10AXIS_typ; (*Zugstation 1*)
	gPBS2 : ACP10AXIS_typ; (*Zugstation 1*)
	gCatchBelt : ACP10AXIS_typ; (*Fangband*)
	gConvBelt : ACP10AXIS_typ; (*Auslageband*)
	gUnwOp : ACP10AXIS_typ; (*Abwickler Operatorseite*)
	gUnwDrv : ACP10AXIS_typ; (*Abwickler Antriebsseite*)
	gBuffer : ACP10AXIS_typ; (*Bahnspeicher*)
	gGridFeeder : ACP10AXIS_typ; (*Drehvorrichtung Gitterturm*)
	gLongCut : ACP10AXIS_typ; (*Drehvorrichtung Gitterturm*)
	gUnwFeeder : ACP10AXIS_typ;
	gUnwFeeder_HW : SdcHwCfg_typ := (0);
	gUnwFeeder_DrvIf : SdcDrvIf16_typ := (0);
	gUnwFeeder_DiDoIf : SdcDiDoIf_typ := (0);
	gUnwFeeder_ModuleOk : BOOL := 0; (* 	gLamPB : ACP10AXIS_typ; ZUgstation der Lamieniereinheit 08.01.14
	gPower : ACP10AXIS_typ;
	gCut3 : ACP10AXIS_typ;
	gTWindTop : ACP10AXIS_typ;
	gTWindBot : ACP10AXIS_typ;
	gPBU : ACP10AXIS_typ;
	gLabelVax : ACP10VAXIS_typ;
	gLabelPBS : ACP10AXIS_typ;
	gConvB : ACP10AXIS_typ;
	gTopBelt : ACP10AXIS_typ;
	gLaminator : ACP10AXIS_typ;
	gLaminator_HW : SdcHwCfg_typ := (0);
	gLaminator_DrvIf : SdcDrvIf16_typ := (0);
	gLaminator_DiDoIf : SdcDiDoIf_typ := (0);
	gLaminator_ModuleOk : BOOL := 0;
	gSpender : ACP10AXIS_typ;
	gSpender_HW : SdcHwCfg_typ := (0);
	gSpender_DrvIf : SdcDrvIf16_typ := (0);
	gSpender_DiDoIf : SdcDiDoIf_typ := (0);
	gSpender_ModuleOk : BOOL := 0;
	Flash_400 : BOOL;
	Cut_unit2_ready_to_ref : BOOL;
	Cut_unit1_ready_to_ref : BOOL;
	Flash_200 : BOOL;
	gLamAufw : ACP10AXIS_typ;
	gLamAufw_HW : SdcHwCfg_typ := (0);
	gLamAufw_DrvIf : SdcDrvIf16_typ := (0);
	gLamAufw_DiDoIf : SdcDiDoIf_typ := (0);
	gLamAufw_ModuleOk : BOOL := 0;
	gAxis01 : ACP10AXIS_typ;
	gAxis02 : ACP10AXIS_typ;*)
END_VAR
(*CONST_MACHINE_MODES_STR : CONST_MACHINE_MODES;*)
VAR
	gAxis03 : ACP10AXIS_typ;
	gAxis03_HW : SdcHwCfg_typ := (0);
	gAxis03_DrvIf : SdcDrvIf16_typ := (0);
	gAxis03_DiDoIf : SdcDiDoIf_typ := (0);
	gAxis03_ModuleOk : BOOL := 0;
	RegMarkControl : ARRAY[0..MAX_RM_AXIS_INDEX] OF reg_mark_typ; (*control structure*)
	AxisRmRef : ARRAY[0..MAX_RM_AXIS_INDEX] OF UDINT; (*array that contains pointer to axis data structure*)
	AxisRmMasterRef : ARRAY[0..MAX_RM_AXIS_INDEX] OF UDINT; (*array that contains pointer to the data structure of the master for the axis*)
	AxisRmCorrRef : ARRAY[0..MAX_RM_AXIS_INDEX] OF UDINT; (*array that contains pointer to axis data structure for correction movement*)
	CutUnit1 : Cut_Type;
	RegMarkIf : RmIf_Type;
	gPackBelt : ACP10AXIS_typ;
	gPackBelt_HW : SdcHwCfg_typ := (0);
	gPackBelt_DrvIf : SdcDrvIf16_typ := (0);
	gPackBelt_DiDoIf : SdcDiDoIf_typ := (0);
	gPackBelt_ModuleOk : BOOL := 0;
END_VAR
```

### GlobConst.var - Package variables
```iecst
(********************************************************************
 * COPYRIGHT -- Bernecker + Rainer
 ********************************************************************
 * File: GlobConst.var
 * Author: schoenefeldr
 * Created: July 18, 2012
 *
 * History:
 *
 * 2012-09-11 /schoenefeldr/
 *    - Renamed additional winder to spender 3
 ********************************************************************
 * Global variables of project 120706_hp_001
 ********************************************************************)
(*======================================================================================================================================*)
(*Recipe constants, e.g. operating modes*)
(*======================================================================================================================================*)
(*Unwinding operating modes*)
VAR CONSTANT
	OPM_UNWINDING_OFF : USINT := 0;
	OPM_UNWINDING_ON : USINT := 1;
END_VAR
VAR CONSTANT
	STATE_READY 		: USINT := 10;
	STATE_POWER_ON	 	: USINT := 1;
	STATE_MOVE_VELOCITY : USINT := 16;
	STATE_MOVE_ABSOLUTE : USINT := 14;
	STATE_WAIT 			: USINT := 0;
	STATE_STOP 			: USINT := 11;
	STATE_MOVE_ADDITIVE : USINT := 15;
	STATE_HOME 			: USINT := 2;
	STATE_ERROR_RESET 	: USINT := 102;
	STATE_ERROR_AXIS 	: USINT := 100;
	STATE_ERROR 		: USINT := 101;
	STATE_JOG_POSITIVE 	: USINT := 12;
	STATE_JOG_NEGATIVE 	: USINT := 13;
	STATE_HALT 			: USINT := 17;
END_VAR
(*Long cut unit operating modes*)
VAR CONSTANT
	OPM_LONG_CUT_DISABLED : UDINT := 10; (*Long cut enabled*)
	OPM_LONG_CUT_ENABLED : UDINT := 11; (*active braking*)
END_VAR
(*Winder operating modes*)
VAR CONSTANT
	OPM_WIND_DISABLED : UDINT := 35; (*Winder disabled*)
	OPM_WIND_WINDER : UDINT := 36; (*Machine ready for operation*)
	OPM_WIND_BRAKE : UDINT := 37; (*Brake functionality*)
END_VAR
(*Web tension unit operating mode*)
VAR CONSTANT
	OPM_WEB_TENSION_DISABLED : UDINT := 5; (*Web tension control disabled*)
	OPM_WEB_TENSION_ENABLED : UDINT := 6; (*Web tension control enabled*)
END_VAR
(*End module operating mode*)
VAR CONSTANT
	OPM_END_MODULE_DISABLED : UDINT := 40; (*No end module selected, disable winder and belts*)
	OPM_END_MODULE_TOP_WINDER : UDINT := 41; (*Select top winder*)
	OPM_END_MODULE_BOT_WINDER : UDINT := 42; (*Select bottom winder*)
	OPM_END_MODULE_TANDEM_WINDER : UDINT := 43; (*Select tandem winder*)
	OPM_END_MODULE_BELTS : UDINT := 44; (*Select upper belt and conveyor belt*)
END_VAR
(*Markpoint operating mode*)
VAR CONSTANT
	OPM_RM_DISABLED : UDINT := 30; (*deactivated*)
	OPM_RM_SENSOR_CONTROL : UDINT := 31; (*Use sensor*)
	OPM_RM_PERIOD_CONTROL : UDINT := 32; (*use period*)
END_VAR
(*Other constants*)
VAR CONSTANT
	MAX_SYNC_PERIODS_INDEX : USINT := 3; (*Highest index on index for sync periods*)
END_VAR
(*======================================================================================================================================*)
(*Axis constants, with attribute comments*)
(*======================================================================================================================================*)
VAR CONSTANT
	AXIS_CUTTING_UNIT1 : USINT := 0; (*Cutting unit 1 (SafeMC, CAM)*)
	AXIS_CUTTING_UNIT2 : USINT := 1; (*Cutting unit 2 (SafeMC, CAM)*)
	AXIS_CUTTING_UNIT3 : USINT := 2; (*Cutting unit 2 (SafeMC, CAM)*)
	AXIS_PULL_BRAKE_ST1 : USINT := 3; (*Pull brake station 1 (CAM)*)
	AXIS_PULL_BRAKE_UNIT : USINT := 4; (*Pull brake unit (CAM)*)
	AXIS_LABEL_PBS : USINT := 5; (*Pull brake station 2 (CAM)*)
	AXIS_LONG_CUT : USINT := 6; (*Long cut unit (SafeMC, CAM)*)
	AXIS_GRID_WINDER1 : USINT := 7; (*Grid winder 1 (CAM)*)
	AXIS_GRID_WINDER2 : USINT := 8; (*Grid winder 2 (CAM)*)
	AXIS_CONVEYOR_BELT : USINT := 9; (*Conveyor belt (CAM)*)
	AXIS_TOP_BELT : USINT := 10; (*Upper belt (CAM)*)
	AXIS_TOP_TANDEM_WIND : USINT := 11; (*Top tandem winder*)
	AXIS_BOT_TANDEM_WIND : USINT := 12; (*Bottom tandem winder*)
	AXIS_LABEL_PBS_VAX : USINT := 13; (*Pull brake station labeler VAX*)
	AXIS_LAMINATOR : USINT := 14; (*Spender 3 (additional winder)*)
	AXIS_MASTER1 : USINT := 15; (*Global virtual master*)
	AXIS_UNWINDER : USINT := 16; (*Global virtual master*)
	AXIS_SPENDER_WINDER : USINT := 17; (*Spender Aufwickler*)
	AXIS_LAMINATORUNIT : USINT := 18; (* Laminator Unit Zugachse der Laminator Einheit*)
	AXIS_UNDEFINED : USINT := 255; (*Undefined axis index*)
END_VAR
(*Power supply module constants*)
VAR CONSTANT
	PSM_MAIN : USINT := 0; (*Main power supply module*)
END_VAR
(*General axis constants*)
VAR CONSTANT
	NUM_OF_AXES : USINT := 19; (*Total number of servo drives, virtual axes and inverter axes*)
	MAX_AXIS_INDEX : USINT := NUM_OF_AXES-1;
	NUM_OF_SAFEMC_AXES : USINT := 3; (*Number of SafeMC servo drives*)
	MAX_SAFEMC_AXIS_INDEX : USINT := NUM_OF_SAFEMC_AXES-1;
	NUM_OF_CAM_AXES : USINT := 10; (*Number of servo drives with CAM automat functions*)
	MAX_CAM_AXIS_INDEX : USINT := NUM_OF_CAM_AXES-1;
	NUM_OF_PSM : USINT := 1; (*Number of power supply modules*)
	MAX_PSM_INDEX : USINT := NUM_OF_PSM-1; (*Last index entry*)
	AXIS_NAME_LENGTH : USINT := 14; (*String length for axis short names*)
END_VAR
(*======================================================================================================================================*)
(*Global drive attribute definitions*)
(*======================================================================================================================================*)
VAR CONSTANT
	IS_SAFE_AXIS : USINT := 0; (*ACOPOS SafeMC*)
	IS_STD_AXIS : USINT := 1; (*ACOPOS servo drive*)
	IS_ASM_AXIS : USINT := 2; (*ACOPOS with ASM*)
	IS_INVERTER_AXIS : USINT := 3; (*ACOPOSinverter*)
	IS_VIRTUAL_AXIS : USINT := 4; (*ACOPOS virtual axis*)
	RETURNS_MTEMP : USINT := 16; (*Returns a motor temperature*)
	RETURNS_TORQUE : USINT := 17; (*Returns a torque value*)
	NEEDS_DIRECT_ERR_ACK : USINT := 18; (*Needs explicit error acknoledge (ACOPOSinverter)*)
	USES_CAM_AUTOMAT : USINT := 19; (*Uses cam automat instead of simple gear functions*)
	USES_CAM_ADD_ELEMENT : USINT := 20; (*Uses cam automat with additive element*)
	HAS_SETPOINT_HZ : USINT := 21; (*Axis with setpoint in user unit Hz (not in µm/s)*)
	HAS_RM_INPUT : USINT := 22; (*Axis with registration mark sensor at trigger input*)
	USES_RM_CONTROL : USINT := 23; (*Uses registration mark control functionality*)
END_VAR
(*Global configuration definitions*)
VAR CONSTANT
	IS_AVAIL : USINT := 0; (*Axis (of any type) is available, i.e. the motor is physically available*)
	IS_ACTIVE : USINT := 1; (*Axis (of any type) is active, i.e. will be enabled*)
	SET_INACTIVE : USINT := 2; (*Axis (of any type) is active yet and must be disabled*)
	SET_ACTIVE : USINT := 3; (*Axis (of any type) is not active yet and must be enabled*)
	IS_MOUNTED : USINT := 4; (*Axis (of any type) is mounted, i.e. the ACOPOS is physically available*)
END_VAR
(*Validation of permanently stored data*)
VAR CONSTANT
	END_OF_PERM_DATA : UDINT := 2769156954; (*Constant for ckeck validity of permanent memory range*)
END_VAR
(*======================================================================================================================================*)
(*Registration mark control*)
(*======================================================================================================================================*)
VAR CONSTANT
	AXIS_RM_CUTTING_UNIT1 : USINT := 0; (*Registration mark at cutting unit 1 *)
	AXIS_RM_CUTTING_UNIT2 : USINT := 1; (*Registration mark at cutting unit 2*)
	NUM_OF_RM_AXES : USINT := 2; (*Total number of servo drives with registration mark control functionalty*)
	MAX_RM_AXIS_INDEX : USINT := NUM_OF_RM_AXES-1;
	NUM_OF_RM_SENSORS : USINT := 2; (*Total number registration mark sensors, may differ from number of regsitration mark axes*)
	MAX_RM_SENSORS_INDEX : USINT := NUM_OF_RM_SENSORS-1;
	SIZE_OF_RM_DATA_ARRAY : USINT := 20; (*Total number of entries for RM data (lines)*)
	MAX_RM_DATA_ARRAY_INDEX : USINT := SIZE_OF_RM_DATA_ARRAY-1;
END_VAR
(*======================================================================================================================================*)
(*Other constants*)
VAR CONSTANT
		CTRL_FIRST_START: 		INT := 0;
		CTRL_GETMODE: 			INT := 1;
		CTRL_SETMODE: 			INT := 2;
		CTRL_SETSTATEAFTER: 	INT := 3;
		CTRL_MANUAL_BEFORE:		INT := 10;
		CTRL_MANUAL:			INT := 11;
		CTRL_MANUAL_AFTER: 		INT := 12;
		CTRL_AUTO_BEFORE: 		INT := 20;
		CTRL_AUTO: 				INT := 22;
		CTRL_AUTO_AFTER: 		INT := 23;
		CTRL_PRODUCTION_BEFORE: INT := 30;
		CTRL_PRODUCTION: 		INT := 32;
		CTRL_PRODUCTION_AFTER: 	INT := 33;
		CTRL_STOP_BEFORE:		INT := 50;
		CTRL_STOP:				INT := 51;
		CTRL_STOP_AFTER:		INT := 52;
		CTRL_RESET_START: 		INT := 75;
		CTRL_RESET: 			INT := 76;
		CTRL_RESET_AFTER: 		INT := 77;
		CTRL_SAFETYSTOP_BEFORE: INT := 82;
		CTRL_SAFETYSTOP: 		INT := 85;
		CTRL_SAFETYSTOP_AFTER: 	INT := 86;
		CTRL_EMERGENCYSTOP_BEFORE: 	INT := 90;
		CTRL_EMERGENCYSTOP_BEFORE1: INT := 91;
		CTRL_EMERGENCYSTOP: 		INT := 92;
		CTRL_EMERGENCYSTOP_AFTER: 	INT := 93; (* Machine modes*)

END_VAR
(*======================================================================================================================================*)
(*Constants for page selection in visualisation*)
VAR CONSTANT
	CHANGE_PAGE_COMPLETE : UINT := 65535;
END_VAR
(*Scaling constants*)
VAR CONSTANT
	SCALE_10V_TO_PERCENT : REAL := (100.0/32767.0); (*10.0 V = 100 %; 10.0 V = 32767*)
	SCALE_DMS_TO_N : REAL := (36.2/33500.0); (*input value of 100.000 corresponds to 100 N with an error of 1.5 % due to 19° angle*)
	SCALE_10V_TO_KN : REAL := (10.0/32767.0); (*10.0 V = 10 kN; 10.0 V = 32767*)
	SCALE_10V_TO_MM : REAL := (1000.0/32767.0); (*10.0 V = 1000 mm; 10.0 V = 32767*)
	SCALE_10V_TO_NM : REAL := (10.0/32767.0); (*10.0 V = 10.0 Nm; 10.0 V = 32767*)
	SCALE_10V_TO_INT : REAL := (32767.0/10.0); (*32767 = 10.0 V, used for min/max calculation*)
END_VAR
```

### GlobMachConst.var - Package variables
```iecst
(********************************************************************
 * COPYRIGHT -- Bernecker + Rainer
 ********************************************************************
 * File: GlobMachConst.var
 * Author: schoenefeldr
 * Created: August 01, 2012
 ********************************************************************
 * Global variables of project 120801_hp_004
 ********************************************************************)
(*======================================================================================================================================*)
(*MACHINE CONSTANTS*)
(*======================================================================================================================================*)
VAR CONSTANT
	MACHINE_WINDCORE_MAXSENSOR : REAL := 995.0; (*995.0 mm maximum sensor value*)
	MACHINE_WINDCORE_MINSENSOR : REAL := 5.0; (*5.0 mm minimum sensor value*)
	MACHINE_WINDCORE_DIAM : REAL := 76.0; (*76 mm diameter winding core*)
	MACHINE_LENGTH_PER_TOOTH : REAL := 3175.0; (*3.175 mm per tooth [µm]*)
	MACHINE_UNITS_PER_METER : REAL := 1000000.0; (*conversion between m and unit, here µm*)

END_VAR
(*Helping constants for linearisation of distance sensors (offline calculated during first setup)*)
VAR CONSTANT
	DIAM_SENSOR_LINEAR_CORR_GAIN : REAL := 0.88105; (*Gain for linear correction of value [1]*)
	DIAM_SENSOR_LINEAR_CORR_OFFSET : REAL := 104.0; (*Offset for linear correction of value [mm]*)

END_VAR
(*Configuration constants*)
VAR CONSTANT
	CFG_FLENGE_DMS_AIN : USINT := 10; (*Binary 1010 for 1000 samples per second*)
END_VAR
(*======================================================================================================================================*)
(*MOVEMENT RELATED MACHINE CONSTANTS*)
(*======================================================================================================================================*)
(*Diese Konstantendefinitionen evtl. verschieben*)
VAR CONSTANT
	GEAR_RATIO_CUT1 : UINT := 5; (*gear ratio of cutting unit gearbox*)
	VELOCITY_LIMIT_OVER_MAX : REAL := 4000000.0; (*Maximum velocity incl. reserve, e.g. 4.000.000 = 240 m/min*)
	MASTER_VELOCITY_INCREMENT : REAL := (1000000.0/60.0); (*default increment/decrement = 1 m/min*)
	MASTER_VELOCITY_HOLD_THRESHOLD : REAL := (1.2*1000000.0/60.0); (*additive velo setpoint for hold/inc cmd (avoid deceleration)*)
	MASTER_VELOCITY_DEC_THRESHOLD : REAL := (0.8*1000000.0/60.0); (*additive velo setpoint for decrement cmd*)
	DEFAULT_MASTER_MAX_VELO : REAL := 1000000.0; (*default maximum velocity e.g. 1.000.000 = 60 m/min*)
	DEFAULT_MASTER_AUTO_MODE_ACC : REAL := (1000000.0/60.0); (*default acceleration e.g. 16666 = 1 (m/min)/s*)
	EMCY_STOP_MASTER_DEC : REAL := 2800000.0; (*master deceleration in case of emergency stop [units/s^2]*)
	EMCY_DOORS_MASTER_DEC : REAL := 1200000.0; (*master deceleration in case of emergency doors opened [units/s^2]*)
	SLS_MASTER_VELO : REAL := 66666.67; (*master velocity in case of Safe Limited Speed [units/s]*)
	DEFAULT_NUMERATOR_DINT : DINT := 10000; (*Default numerator for electronic gear (CAM or Gear)*)
	DEFAULT_DENOMINATOR_UDINT : UDINT := 10000; (*Default denominator for electronic gear (CAM or Gear)*)
	DEFAULT_NUMERATOR_REAL : REAL := DEFAULT_NUMERATOR_DINT; (*Default numerator for electronic gear (CAM or Gear)*)
	DEFAULT_DENOMINATOR_REAL : REAL := DEFAULT_DENOMINATOR_UDINT; (*Default denominator for electronic gear (CAM or Gear)*)
	MAX_VELO_REL_10_PERCENT : REAL := 10.0; (*maximum relative value [%], 100 = 100 %*)
	GEAR_RATIO_TOP_TWIND : REAL := 3600.0/484.0; (*gear ratio of top tandem winder from toothbelt gear*)
	GEAR_RATIO_BOT_TWIND : REAL := 3600.0/484.0; (*gear ratio of bottom tandem winder from toothbelt gear*)
	GEAR_RATIO_UNWINDER : REAL := 8.0;
	MAX_CORRECTION : REAL := 3000.0;
END_VAR
(*======================================================================================================================================*)
(*DEFAULT RECIPE VALUES (MACHINE AND APPLICATION)*)
(*======================================================================================================================================*)
VAR CONSTANT
	DEFAULT_TWIND_WARN_DIAM : REAL := 500.0; (*Default warning diameter tandem winder [mm]*)
	DEFAULT_TWIND_STOP_DIAM : REAL := 600.0; (*Default stop diameter tandem winder [mm]*)
	DEFAULT_TOP_TWIND_FRICT_COMP : REAL := 0.25; (*Default friction compensation top tandem winder [Nm] (on motor side)*)
	DEFAULT_BOT_TWIND_FRICT_COMP : REAL := 0.25; (*Default friction compensation bottom tandem winder [Nm] (on motor side)*)
	DEFAULT_LOAD_UNITS_80 : UDINT := 50800000; (*Default encoder_if - scaling - load units for number of teeth = 80*)
	DEFAULT_LOAD_REV_MOTOR_200 : UDINT := 1000; (*Default encoder_if - scaling - load - motor_rev for number of teeth = 200*)
	DEFAULT_COG_SUPP_SPINDLE : UINT := 160; (*Default number of teeth of cog support spindle*)
	DEFAULT_COG_TOOL_SEGMENTS : USINT := 1; (*Default number of teeth of cog cutting*)
	DEFAULT_COG_CUTTING : UINT := 96; (*Default number of teeth of cog cutting*)
	DEFAULT_TWIND_MIN_DIAM_FORCE : REAL := 10.0; (*Default winder force (tandem winder) at low diameter*)
	DEFAULT_TWIND_MAX_DIAM_FORCE : REAL := 5.0; (*Default winder force (tandem winder) at stop diameter*)
	DEFAULT_TWIND_MIN_DIAM_VAL : REAL := 100000.0; (*Default value for low diameter [µm]*)
END_VAR
(*======================================================================================================================================*)
(*OTHER CONSTANTS*)
(*======================================================================================================================================*)
(*Time delay values*)
VAR CONSTANT
	DELAY_DRIVE_ENABLE : TIME := T#15s; (*Delay [ms] until the drives are enabled by software*)
	DELAY_REQUEST_STO : TIME := T#1s850ms; (*Delay [ms] until the drives have to be disabled if STO is requested*)
	TIMEOUT_START : UINT := 1000; (*Timeout [ms] for checking if the active drive ar in the proper axis state (PLCopen)*)
END_VAR
```
